# B&R Automation Studio project Panasonic_LinkaPowerCP2_A2021055 (part 4)

### Global.typ - Global data types
```iecst
(********************************************************************
 * COPYRIGHT -- Microsoft
 ********************************************************************
 * File: Global.typ
 * Author: Martin
 * Created: February 11, 2016
 ********************************************************************
 * Global data types of project Zamazat_1
 ********************************************************************)
(*************Vizualizacia******************************)

TYPE
	P1_Vizu_typ : 	STRUCT
		ActualPage : STRING[80];
		GoPage : STRING[80] := 'PageBootP1';
		TL_ResetCS : BOOL;
		TL_RezimAutomat : BOOL;
		ZobrazHL1_ST1 : BOOL; (*ST1 - Chýbajúci material na paletke 4F*)
		ZobrazHL2_ST1 : BOOL; (*ST1 - Chýbajúci material na paletke 5F*)
		ZobrazHL3_ST1 : BOOL; (*ST1 - Chýbajúci material na paletke 5H*)
		ZobrazHL4_ST1 : BOOL; (*ST1 - Zlý alebo neprečítaný QR kód na Power CP*)
		ZobrazHL5_ST1 : BOOL; (*ST1 - Zle zacvaknuté alebo chýbajúce piny DPS*)
		ZobrazHL6_ST1 : BOOL; (*ST1 - Zlý alebo neprečítaný QR kód DPS*)
		ZobrazHL7_ST1 : BOOL; (*ST1 - Nesprávny QR kód Power CP*)
		ZobrazHL8_ST1 : BOOL; (*ST1 - Nesprávny QR kód DPS*)
		ZobrazHL9_ST1 : BOOL; (*ST1 - Odpoved systemu tracebility je NG*)
		ZobrazHL10_ST1 : BOOL;
		ZobrazHL11_ST1 : BOOL;
		ZobrazHL12_ST1 : BOOL;
		ZobrazHL13_ST1 : BOOL;
		ZobrazHL14_ST1 : BOOL; (*ST1 - Nieje prihlásený operátor*)
		ZobrazHL15_ST1 : BOOL; (*ST1 - Panatrace neodpovedá*)
		ZobrazHL1_ST2 : BOOL;
		ZobrazHL2_ST2 : BOOL;
		ZobrazHL3_ST2 : BOOL;
		ZobrazHL4_ST2 : BOOL;
		ZobrazHL5_ST2 : BOOL;
		ZobrazHL6_ST2 : BOOL;
		ZobrazHL7_ST2 : BOOL;
		ZobrazHL8_ST2 : BOOL;
		ZobrazHL9_ST2 : BOOL; (*ST2 - Odpoved panatrace NG*)
		ZobrazHL10_ST2 : BOOL; (*ST2 - Panatrace neodpovedá*)
		TL_PrednyZamok_Farba : WSTRING[80];
		TL_ZadnyZamok_Farba : WSTRING[80];
		TL_ZamkniPrednyZamok : BOOL;
		TL_ZamkniZadnyZamok : BOOL;
		TL_StartAutomat_ENABLE : BOOL;
		TL_KoniecCyklu_ENABLE : BOOL;
		TL_Uzivatelia_ENABLE : BOOL;
		TL_STOP_ENABLE : BOOL;
		TL_SETUP_ENABLE : BOOL;
		TL_VyprazdnenieLinky_ENABLE : BOOL;
		TL_RezimAutomat_ENABLE : BOOL;
		TL_RezimManual_ENABLE : BOOL;
		TL_OvladaniaZamkov_ENABLE : BOOL;
		TL_VolbaModelu_ENABLE : BOOL;
		TL_PaletkaPrechadza_ENABLE : BOOL;
		TL_TestovaciKus_ENABLE : BOOL;
		TL_Revork_ENABLE : BOOL;
		TL_OvladanieVytahu_ENABLE : BOOL;
		TL_PrihlasenieOperatora_ENABLE : BOOL;
		TL_PrihlasovOperatora_AKTIVNE : BOOL;
		TL_VycistiSkrutkovackuK30_ENABLE : BOOL;
		TL_PolohujManipulator_ENABLE : BOOL;
		Tl_VysunutieSkrutkovK30_ENABLE : BOOL;
		TL_OvladaniaVysunSkrutkovM4_M5 : BOOL;
		TL_OvladSkrutkovSetuK30_ENABLE : BOOL;
		TL_OvladManipulatoraXY_ENABLE : BOOL;
		Srobovanie_OvlManipOsX_ENABLE : BOOL;
		Srobovanie_OvlManipOsY_ENABLE : BOOL;
		EditaciaParametrov_ENABLE : BOOL;
		RR_CistenieSkrutkovaciek_ENABLE : BOOL;
		RR_PozicieSkrutiek_ENABLE : BOOL;
		Vytah_CitaniePaletky_ENABLE : BOOL;
		Vytah_ZapisPaletky_ENABLE : BOOL;
		Warnings_Farba : WSTRING[80];
		Warnings_Index : USINT;
		IndexStavu_Dopravnik : USINT;
		IndexStavu_Vytah : USINT;
		IndexStavu_SpodnyStoper : USINT;
		IndexStavu_StoperSrobovania : USINT;
		IndexStavu_Srobovanie : USINT;
		IndexStavu_AkumulacnyStoper : USINT;
		IndexStavu_Robot : USINT;
	END_STRUCT;
	P2_Vizu_typ : 	STRUCT
		ActualPage : STRING[80];
		GoPage : STRING[80] := 'PageBootP2';
		TL_RezimAutomat : BOOL;
		TL_PrednyZamok_Farba : WSTRING[80];
		TL_ZadnyZamok_Farba : WSTRING[80];
		TL_ZamkniPredneZamky : BOOL;
		TL_ZamkniZadneZamky : BOOL;
		TL_StartAutomat_ENABLE : BOOL;
		TL_KoniecCyklu_ENABLE : BOOL;
		TL_STOP_ENABLE : BOOL;
		TL_SETUP_ENABLE : BOOL;
		TL_RezimAutomat_ENABLE : BOOL;
		TL_RezimManual_ENABLE : BOOL;
		TL_RRZdvihZaklTesnenia_ENABLE : BOOL;
		TL_RRPojazdZaklTesnenia_ENABLE : BOOL;
		TL_OvladaniaZamkov_ENABLE : BOOL;
		TL_VycistiSkrutkovackuM6_ENABLE : BOOL;
		TL_VycistiSkrutkovackuM5_ENABLE : BOOL;
		TL_PolohujManipulator_ENABLE : BOOL;
		TL_VysunutiaMaticovacM4_ENABLE : BOOL;
		Tl_VysunutieSkrutkovM6_ENABLE : BOOL;
		Tl_VysunutieSkrutkovM5_ENABLE : BOOL;
		TL_OvladaniaVysunSkrutkovM4 : BOOL;
		TL_OvladManipulatoraXY_ENABLE : BOOL;
		TL_OvladSkrutkovSetuM6_ENABLE : BOOL;
		TL_OvladSkrutkovSetuM5_ENABLE : BOOL;
		TL_PresunZvarania_ENABLE : BOOL;
		TL_ZdvihZvarania_ENABLE : BOOL;
		TL_StartSekvencieZvarania_ENABLE : BOOL;
		EditaciaParametrov_ENABLE : BOOL;
		ZaklTesnenia_OvlZdvihu_ENABLE : BOOL;
		ZaklTesnenia_OvlZostupu_ENABLE : BOOL;
		ZaklTesnenia_OvlPojazdu_ENABLE : BOOL;
		Srobovanie_OvlManipOsX_ENABLE : BOOL;
		Srobovanie_OvlManipOsY_ENABLE : BOOL;
		Zvaranie_OvlZdvihu_ENABLE : BOOL;
		RR_CistenieSkrutkovaciek_ENABLE : BOOL;
		RR_PozicieSkrutiek_ENABLE : BOOL;
		TL_PrihlasenieOperatora_ENABLE : BOOL;
		TL_PrihlasovOperatora_AKTIVNE : BOOL;
		TL_ResetCS : BOOL;
		Warnings_Farba : WSTRING[80];
		Warnings_Index : USINT;
		StavPracoviska_Index : USINT;
		ZobrazPopUp_0 : BOOL;
		ZobrazPopUp_1 : BOOL;
		ZobrazPopUp_2 : BOOL;
		PopUpButtonYES : BOOL;
		PopUpButtonNO : BOOL;
		ZobrazHL1_ST3 : BOOL; (*ST3 - Chýbajúci material na paletke 4F *)
		ZobrazHL2_ST3 : BOOL; (*ST3 - Chýbajúci material na paletke 5F*)
		ZobrazHL3_ST3 : BOOL; (*ST3 - Chýbajúci material na paletke 5H*)
		ZobrazHL4_ST3 : BOOL; (*ST3 - Skontroluj prítomnosť alebo QR kód filtra 5H*)
		ZobrazHL5_ST3 : BOOL; (*ST3 - V zakladači chýba Power CP !!!*)
		ZobrazHL6_ST3 : BOOL; (*ST3 - V zakladači chýba tesnenie !!!*)
		ZobrazHL7_ST3 : BOOL; (*ST3 - Zle založené tesnenie na Power CP*)
		ZobrazHL8_ST3 : BOOL; (*ST3 - Založenie tesnenia je OK, odober Power CP zo zakladača *)
		ZobrazHL9_ST3 : BOOL; (*ST3 - Nesprávny QR kód filtra 5H*)
		ZobrazHL10_ST3 : BOOL; (*ST3 - Nesprávny alebo neprečítaný QR kód Power CP*)
		ZobrazHL11_ST3 : BOOL; (*ST3 - Odpoved systemu tracebility je NG*)
		ZobrazHL12_ST3 : BOOL; (*ST3 - Operátor nieje prihlásený*)
		ZobrazHL13_ST3 : BOOL; (*ST3 - Odpoved panatrace je NG*)
		ZobrazHL14_ST3 : BOOL; (*ST3 - Odober PowerCP z paletky a vlož do šuplíka*)
		ZobrazHL15_ST3 : BOOL; (*ST3 - Panatrace neodpovedá*)
		ZobrazHL1_ST4 : BOOL;
		ZobrazHL2_ST4 : BOOL;
		ZobrazHL3_ST4 : BOOL; (*ST4 -Odpoved panatrace je NG*)
		ZobrazHL4_ST4 : BOOL; (*ST4 - Panatrace neodpovedá*)
		ZobrazHL1_ST5 : BOOL;
		ZobrazHL2_ST5 : BOOL;
		ZobrazHL3_ST5 : BOOL;
		ZobrazHL4_ST5 : BOOL; (*ST5 - Odpoved panatrace je NG*)
		ZobrazHL5_ST5 : BOOL; (*ST5 - Model 4F kontrola skrutiek M4 s komaxitom*)
		ZobrazHL6_ST5 : BOOL; (*ST5 - Model 5F kontrola skrutiek M4 s komaxitom*)
		ZobrazHL7_ST5 : BOOL; (*ST5 - Model 5H kontrola skrutiek M4 bez komaxitu*)
		ZobrazHL8_ST5 : BOOL; (*ST5 - Panatrace neodpovedá*)
		ZobrazHL1_ST6 : BOOL; (*ST6 - Chýbajúci material na paletke 4F *)
		ZobrazHL2_ST6 : BOOL; (*ST6 - Chýbajúci material na paletke 5F*)
		ZobrazHL3_ST6 : BOOL; (*ST6 - Chýbajúci material na paletke 5H*)
		ZobrazHL4_ST6 : BOOL; (*ST6 - Skontroluj prítomnosť alebo QR kód filtra 5H*)
		ZobrazHL5_ST6 : BOOL; (*ST6 - V zakladači chýba Power CP !!!*)
		ZobrazHL6_ST6 : BOOL; (*ST6 - V zakladači chýba tesnenie !!!*)
		ZobrazHL7_ST6 : BOOL; (*ST6 - Zle založené tesnenie na Power CP*)
		ZobrazHL8_ST6 : BOOL; (*ST6 - Odpoved panatrace je NG*)
		ZobrazHL9_ST6 : BOOL; (*ST6 - Panatrace neodpovedá*)
		IndexStavu_Dopravnik : USINT;
		IndexStavu_SpodnyStoper : USINT;
		IndexStavu_StoperZakladacaTesn : USINT;
		IndexStavu_ZakladacaTesnenia : USINT;
		IndexStavu_StoperMaticovacky : USINT;
		IndexStavu_AkumulacnyStoper : USINT;
		IndexStavu_StoperSrobovania : USINT;
		IndexStavu_Srobovania : USINT;
		IndexStavu_Robot : USINT;
		IndexStavu_StoperZvarania : USINT;
		IndexStavu_Zvaranie : USINT;
		IndexStavu_Cistenie : USINT;
	END_STRUCT;
	P34_Vizu_typ : 	STRUCT
		ActualPage : STRING[80];
		GoPage : STRING[80] := 'PageBootP34';
		TL_RezimAutomat : BOOL;
		ZobrazHL1_ST7 : BOOL; (*ST7 - Odpoved panatrace je NG*)
		ZobrazHL2_ST7 : BOOL; (*ST7 - Panatrace neodpovedá*)
		ZobrazHL1_ST8 : BOOL; (*ST8A - Odpoved panatrace je NG*)
		ZobrazHL2_ST8 : BOOL; (*ST8B - Odpoved panatrace je NG*)
		ZobrazHL3_ST8 : BOOL; (*ST8A - Panatrace neodpovedá*)
		ZobrazHL4_ST8 : BOOL; (*ST8B - Panatrace neodpovedá*)
		ZobrazHL1_ST9 : BOOL;
		ZobrazHL2_ST9 : BOOL;
		ZobrazHL3_ST9 : BOOL; (*ST9 - Odpoved panatrace je NG*)
		ZobrazHL4_ST9 : BOOL; (*ST9 - Panatrace neodpovedá*)
		ZobrazHL1_ST10 : BOOL; (*ST10 - Chýbajúci material na paletke 4F *)
		ZobrazHL2_ST10 : BOOL; (*ST10 - Chýbajúci material na paletke 5F*)
		ZobrazHL3_ST10 : BOOL; (*ST10 - Chýbajúci material na paletke 5H*)
		ZobrazHL4_ST10 : BOOL; (*ST10 - Paletka nieje prázdna*)
		ZobrazHL5_ST10 : BOOL; (*ST10 - Paletka nieje prázdna*)
		ZobrazHL6_ST10 : BOOL; (*ST10 - Paletka nieje prázdna*)
		ZobrazHL7_ST10 : BOOL; (*ST10 - Nieje prihlaseny operator*)
		ZobrazHL8_ST10 : BOOL;
		ZobrazHL9_ST10 : BOOL; (*ST10 - Odpoved panatrace je NG*)
		ZobrazHL10_ST10 : BOOL; (*ST10 - Panatrace neodpovedá*)
		ZobrazHL1_HVtest : BOOL; (*HV tester neodpovedá*)
		ZobrazHL1_FinalTestA : BOOL; (*Final tester neodpovedá*)
		ZobrazHL1_FinalTestB : BOOL; (*Final tester neodpovedá*)
		TL_ResetCS : BOOL;
		IndexStavu_DopravnikP3 : USINT;
		IndexStavu_SpodnyStoperP3 : USINT;
		IndexStavu_StoperSrobovaniaP3 : USINT;
		IndexStavu_SrobovanieP3 : USINT;
		IndexStavu_HV_Test : USINT;
		IndexStavu_AkumulacnyStoperP3 : USINT;
		IndexStavu_ZdvizkPredLeakTestomA : USINT;
		IndexStavu_ZdvizkPredLeakTestomB : USINT;
		IndexStavu_StoperLeakageTestA : USINT;
		IndexStavu_StoperLeakageTestB : USINT;
		IndexStavu_ZdvizkaZaLeakTestomA : USINT;
		IndexStavu_ZdvizkaZaLeakTestomB : USINT;
		IndexStavu_DopravnikP4 : USINT;
		IndexStavu_SpodnyStoperP4 : USINT;
		IndexStavu_Vytah : USINT;
		IndexStavu_StoperFunkcnyTestA : USINT;
		IndexStavu_StoperFunkcnyTestB : USINT;
		IndexStavu_ZdvizkaZaFunkTestomA : USINT;
		IndexStavu_ZdvizkaZaFunkTestomB : USINT;
		IndexStavu_StoperEtiketovackyP4 : USINT;
		TL_PrednyZamok_Farba_P3 : WSTRING[80];
		TL_ZadnyZamok_Farba_P3 : WSTRING[80];
		TL_ZamkniPredneZamky_P3 : BOOL;
		TL_ZamkniZadneZamky_P3 : BOOL;
		TL_StartAutomat_ENABLE_P3 : BOOL;
		TL_KoniecCyklu_ENABLE_P3 : BOOL;
		TL_STOP_ENABLE_P3 : BOOL;
		TL_SETUP_ENABLE : BOOL;
		TL_RezimAutomat_ENABLE : BOOL;
		TL_RezimManual_ENABLE_P3 : BOOL;
		TL_RezimManual_ENABLE_P4 : BOOL;
		TL_OvladaniaZamkov_ENABLE_P3 : BOOL;
		TL_OvladaniaZamkov_ENABLE_P4 : BOOL;
		TL_StartAutomat_ENABLE_P4 : BOOL;
		TL_KoniecCyklu_ENABLE_P4 : BOOL;
		TL_STOP_ENABLE_P4 : BOOL;
		TL_VycistiSkrutkovackuK40_ENABLE : BOOL;
		TL_PolohujManipulator_ENABLE : BOOL;
		Tl_VysunutieSkrutkovK40_ENABLE : BOOL;
		TL_OvladaniaVysunSkrutkovM5 : BOOL;
		TL_OvladManipulatoraY_ENABLE : BOOL;
		TL_OvladSkrutkovSetuK40_ENABLE : BOOL;
		TL_SekvencieHV_Testu_ENABLE : BOOL;
		TL_OvladaniaHV_Testu_ENABLE : BOOL;
		TL_SekvencieLeakTestuA_ENABLE : BOOL;
		TL_OvladaniaLeakTestuA_ENABLE : BOOL;
		TL_SekvencieLeakTestuB_ENABLE : BOOL;
		TL_OvladaniaLeakTestuB_ENABLE : BOOL;
		TL_SekvencieFunkcTestuA_ENABLE : BOOL;
		TL_OvladaniaFunkcTestuA_ENABLE : BOOL;
		TL_SekvencieFunkcTestuB_ENABLE : BOOL;
		TL_OvladaniaFunkcTestuB_ENABLE : BOOL;
		TL_SekvencieEtiketovania_ENABLE : BOOL;
		TL_OvladaniaEtiketovania_ENABLE : BOOL;
		TL_ZdvihAplikEtiketovania_ENABLE : BOOL;
		Vytah_CitaniePaletky_ENABLE : BOOL;
		Vytah_ZapisPaletky_ENABLE : BOOL;
		Srobovanie_OvlManipOsY_ENABLE : BOOL;
		VolbaLeakageTestu_ENABLE : BOOL;
		VolbaFunkcnehoTestu_ENABLE : BOOL;
		EditaciaParametrov_ENABLE : BOOL;
		RR_CistenieSkrutkovaciek_ENABLE : BOOL;
		RR_PozicieSkrutiek_ENABLE : BOOL;
		TL_PrihlasenieOperatora_ENABLE : BOOL;
		TL_PrihlasovOperatora_AKTIVNE : BOOL;
		TL_PrednyZamok_Farba_P4 : WSTRING[80];
		TL_ZadnyZamok_Farba_P4 : WSTRING[80];
		TL_ZamkniPrednyZamok_P4 : BOOL;
		TL_ZamkniZadnyZamok_P4 : BOOL;
		WarningsP3_Farba : WSTRING[80];
		WarningsP3_Index : USINT;
		WarningsP4_Farba : WSTRING[80];
		WarningsP4_Index : USINT;
		TL_VyprazdnenieLinky_ENABLE : BOOL;
	END_STRUCT;
	Vizu_typ : 	STRUCT
		TL_ResetCS_Farba : WSTRING[80];
		ZadanyCasPLC : DATE_AND_TIME;
		NastavCasPLC : BOOL;
		AktualnyCasPLC : DATE_AND_TIME;
	END_STRUCT;
END_TYPE

(*************Parametre paletky*********************)

TYPE
	Paletka_typ : 	STRUCT
		PAR : Paletka_PAR_typ; (*Parametre komunikácie z Panatrace*)
		STAV : Paletka_STAV_typ;
	END_STRUCT;
	Paletka_PAR_typ : 	STRUCT
		CisloPaletky : STRING[2]; (*Je pevne dané čipom RFID*)
		QRkodPowerCP : STRING[30]; (*Načítam ho na prvom výťahu a posielam ho na server ako master number *)
		QRkodFiltra_5H : STRING[32]; (*Načítam ho na pracovisku zakladania tesnenia a párujem ho s QR kodom Power CP*)
		QRkodFiltra_4F5F : STRING[32]; (*Načítam ho na prvom výtahu a párujem ho s QR kodom Power CP*)
		ID_Operatora : STRING[80]; (*Číslo karty operátora*)
		StavPowerCP : STRING[4]; (*Stav vyžiadaný zo servera  - PASS, FAIL,  ktorý sa mení v pribehu výroby *)
	END_STRUCT;
	Paletka_STAV_typ : 	STRUCT
		StavPaletky : STRING[10]; (*OK - paletka OK , NG - paletka NG, REV - revork, TEST - testovací kus, PRECH - paletka iba prechádza*)
		TypModelu : STRING[5]; (*4F, 5F, 5H podla zvolenej receptury*)
		KodModelu : STRING[32]; (*Dostanem pridelene na pracovisku etiketovania*)
		CisloTestovacejStanice : STRING[20]; (*Číslo testovacej stanice*)
		CisloRevorkovejStanice : STRING[20]; (*Číslo revorkovej stanice*)
		Zvaranie_Ukoncene : BOOL;
		HV_Test_Ukonceny : BOOL;
		LeakageTest_Ukonceny : BOOL;
		FunkcnyTest_Ukonceny : BOOL;
		QRkodFiltraPriradeny : BOOL;
		NalepenieEtikety_DONE : BOOL;
		OdoslanieFotiek_DONE : BOOL;
		Komunikacia_DONE : BOOL;
		CisloEtiketyVyziadane : BOOL;
	END_STRUCT;
END_TYPE

(*****************Remanentne premenne**********)

TYPE
	P1_RemPremenne_typ : 	STRUCT
		P1_Srob45F_PozX_LavejSkrutkyK30 : REAL;
		P1_Srob45F_PozY_LavejSkrutkyK30 : REAL;
		P1_Srob45F_PozX_PravejSkrutkyK30 : REAL;
		P1_Srob45F_PozY_PravejSkrutkyK30 : REAL;
		P1_Srob4F_PozX_ZadnejSkrutkyM4 : REAL;
		P1_Srob4F_PozY_ZadnejSkrutkyM4 : REAL;
		P1_Srob5F_PozX_ZadnejSkrutkyM4 : REAL;
		P1_Srob5F_PozY_ZadnejSkrutkyM4 : REAL;
		P1_Srob45F_Mom_ZadnejSkrutkyM4 : REAL;
		P1_Srob45F_Rychl_ZadnejSkrutkyM4 : REAL; (*mm/s*)
		P1_Srob4F_PozX_PrednejSkrutkyM4 : REAL;
		P1_Srob4F_PozY_PrednejSkrutkyM4 : REAL;
		P1_Srob5F_PozX_PrednejSkrutkyM4 : REAL;
		P1_Srob5F_PozY_PrednejSkrutkyM4 : REAL;
		P1_Srob45F_Mom_PrednejSkrutkyM4 : REAL;
		P1_Srob45F_Rychl_PredneSkrutkyM4 : REAL; (*mm/s*)
		P1_Srob45F_PozX_SkrutkyDPS_M4 : REAL;
		P1_Srob45F_PozY_SkrutkyDPS_M4 : REAL;
		P1_Srob45F_Mom_SkrutkyDPS_M4 : REAL;
		P1_Srob45F_Rychl_SkrutkyDPS_M4 : REAL; (*mm/s*)
		P1_Srob5H_PozX_LavejSkrutkyK30 : REAL;
		P1_Srob5H_PozY_LavejSkrutkyK30 : REAL;
		P1_Srob5H_PozX_PravejSkrutkyK30 : REAL;
		P1_Srob5H_PozY_PravejSkrutkyK30 : REAL;
		P1_Srob5H_PozX_LavejSkrutkyM5 : REAL;
		P1_Srob5H_PozY_LavejSkrutkyM5 : REAL;
		P1_Srob5H_Mom_LavejSkrutkyM5 : REAL;
		P1_Srob5H_Rychl_LavejSkrutkyM5 : REAL; (*mm/s*)
		P1_Srob5H_PozX_StrednejSkrutkyM5 : REAL;
		P1_Srob5H_PozY_StrednejSkrutkyM5 : REAL;
		P1_Srob5H_Mom_StrednejSkrutkyM5 : REAL;
		P1_Srob5H_Rychl_StredneSkrutkyM5 : REAL; (*mm/s*)
		P1_Srob5H_PozX_PravejSkrutkyM5 : REAL;
		P1_Srob5H_PozY_PravejSkrutkyM5 : REAL;
		P1_Srob5H_Mom_PravejSkrutkyM5 : REAL;
		P1_Srob5H_Rychl_PravejSkrutkyM5 : REAL; (*mm/s*)
		P1_Srob_PozX_OdobratSkrutkyM5 : REAL;
		P1_Srob_PozY_OdobratSkrutkyM5 : REAL;
		P1_Srob_PozZ_OdobratSkrutkyM5 : REAL;
		P1_Srob_PozX_OdobratSkrutkyM4 : REAL;
		P1_Srob_PozY_OdobratSkrutkyM4 : REAL;
		P1_Srob_PozZ_OdobratSkrutkyM4 : REAL;
		P1_Vytah_RychlostZdvihu : REAL; (*mm/s*)
		P1_Vytah_Zdvih_Acc : REAL;
		P1_Vytah_Zdvih_Dcc : REAL;
		P1_Vytah_PoziciaNakladania : REAL;
		P1_Vytah_PoziciaVykladania : REAL;
		P1_ManipSrob_OsX_Rychlost : REAL; (*mm/s*)
		P1_ManipSrob_OsY_Rychlost : REAL; (*mm/s*)
		P1_ManipSrob_OsXY_Acc : REAL;
		P1_ManipSrob_OsXY_Dcc : REAL;
		P1_ManipSrob_OsZ_M4_Rychlost : REAL; (*mm/s*)
		P1_ManipSrob_OsZ_M4_Acc : REAL;
		P1_ManipSrob_OsZ_M4_Dcc : REAL;
		P1_ManipSrob_OsZ_M5_Rychlost : REAL; (*mm/s*)
		P1_ManipSrob_OsZ_M5_Acc : REAL;
		P1_ManipSrob_OsZ_M5_Dcc : REAL;
		P1_Srob45F_LavaK30_Vysunutie_LO : REAL; (*Vysunutie skrutkovačky - spodná tolerancia*)
		P1_Srob45F_LavaK30_Vysunutie_HI : REAL; (*Vysunutie skrutkovačky - horná tolerancia*)
		P1_Srob45F_PravaK30_Vysunutie_LO : REAL; (*Vysunutie skrutkovačky - spodná tolerancia*)
		P1_Srob45F_PravaK30_Vysunutie_HI : REAL; (*Vysunutie skrutkovačky - horná tolerancia*)
		P1_Srob45F_ZadnaM4_Vysunutie_LO : REAL; (*Vysunutie skrutkovačky - spodná tolerancia*)
		P1_Srob45F_ZadnaM4_Vysunutie_HI : REAL; (*Vysunutie skrutkovačky - horná tolerancia*)
		P1_Srob45F_PrednaM4_Vysunutie_LO : REAL; (*Vysunutie skrutkovačky - spodná tolerancia*)
		P1_Srob45F_PrednaM4_Vysunutie_HI : REAL; (*Vysunutie skrutkovačky - horná tolerancia*)
		P1_Srob45F_DPS_M4_Vysunutie_LO : REAL; (*Vysunutie skrutkovačky - spodná tolerancia*)
		P1_Srob45F_DPS_M4_Vysunutie_HI : REAL; (*Vysunutie skrutkovačky - horná tolerancia*)
		P1_Srob5H_LavaK30_Vysunutie_LO : REAL; (*Vysunutie skrutkovačky - spodná tolerancia*)
		P1_Srob5H_LavaK30_Vysunutie_HI : REAL; (*Vysunutie skrutkovačky - horná tolerancia*)
		P1_Srob5H_PravaK30_Vysunutie_LO : REAL; (*Vysunutie skrutkovačky - spodná tolerancia*)
		P1_Srob5H_PravaK30_Vysunutie_HI : REAL; (*Vysunutie skrutkovačky - horná tolerancia*)
		P1_Srob5H_LavaM5_Vysunutie_LO : REAL; (*Vysunutie skrutkovačky - spodná tolerancia*)
		P1_Srob5H_LavaM5_Vysunutie_HI : REAL; (*Vysunutie skrutkovačky - horná tolerancia*)
		P1_Srob5H_StrednaM5_Vysunutie_LO : REAL; (*Vysunutie skrutkovačky - spodná tolerancia*)
		P1_Srob5H_StrednaM5_Vysunutie_HI : REAL; (*Vysunutie skrutkovačky - horná tolerancia*)
		P1_Srob5H_PravaM5_Vysunutie_LO : REAL; (*Vysunutie skrutkovačky - spodná tolerancia*)
		P1_Srob5H_PravaM5_Vysunutie_HI : REAL; (*Vysunutie skrutkovačky - horná tolerancia*)
	END_STRUCT;
	P2_RemPremenne_typ : 	STRUCT
		P2_ZaklTesn_Zdvih_RychlostZdvihu : REAL; (*mm/s*)
		P2_ZaklTesn_Zdvih_RychlZatlacen : REAL; (*mm/s*)
		P2_ZaklTesn_Zdvih_Acc : REAL;
		P2_ZaklTesn_Zdvih_Dcc : REAL;
		P2_ZaklTesn_Zdvih_MomZatlacen : REAL;
		P2_ZaklTesn_Zdvih_PozZatlacenia : REAL;
		P2_ZaklTesn_Pojazd_RychlVysun : REAL;
		P2_ZaklTesn_Pojazd_RychlZasun : REAL;
		P2_ZaklTesn_Pojazd_Acc : REAL;
		P2_ZaklTesn_Pojazd_Dcc : REAL;
		P2_ZaklTesn_Pojazd_PozZatlacenia : REAL;
		P2_ZaklTesn_Pojazd_PozVkladania : REAL;
		P2_ZaklTesn_PocetZatlaceni : USINT;
		P2_Srob4F_PozX_LavejSkrutkyM6 : REAL;
		P2_Srob4F_PozY_LavejSkrutkyM6 : REAL;
		P2_Srob4F_PozX_PravejSkrutkyM6 : REAL;
		P2_Srob4F_PozY_PravejSkrutkyM6 : REAL;
		P2_Srob4F_PozX_LavejSkrutkyM4 : REAL;
		P2_Srob4F_PozY_LavejSkrutkyM4 : REAL;
		P2_Srob45F_Mom_LavejSkrutkyM4 : REAL;
		P2_Srob45F_Rychl_LavejSkrutkyM4 : REAL; (*mm/s*)
		P2_Srob4F_PozX_PravejSkrutkyM4 : REAL;
		P2_Srob4F_PozY_PravejSkrutkyM4 : REAL;
		P2_Srob45F_Mom_PravejSkrutkyM4 : REAL;
		P2_Srob45F_Rychl_PravejSkrutkyM4 : REAL; (*mm/s*)
		P2_Srob5F_PozX_LavejSkrutkyM6 : REAL;
		P2_Srob5F_PozY_LavejSkrutkyM6 : REAL;
		P2_Srob5F_PozX_PravejSkrutkyM6 : REAL;
		P2_Srob5F_PozY_PravejSkrutkyM6 : REAL;
		P2_Srob5F_PozX_LavejSkrutkyM4 : REAL;
		P2_Srob5F_PozY_LavejSkrutkyM4 : REAL;
		P2_Srob5F_PozX_PravejSkrutkyM4 : REAL;
		P2_Srob5F_PozY_PravejSkrutkyM4 : REAL;
		P2_Srob5H_PozX_LavejSkrutkyM5 : REAL;
		P2_Srob5H_PozY_LavejSkrutkyM5 : REAL;
		P2_Srob5H_PozX_PravejSkrutkyM5 : REAL;
		P2_Srob5H_PozY_PravejSkrutkyM5 : REAL;
		P2_Srob5H_PozX_SkrutkyM4 : REAL;
		P2_Srob5H_PozY_SkrutkyM4 : REAL;
		P2_Srob5H_Mom_SkrutkyM4 : REAL;
		P2_Srob5H_Rychl_SkrutkyM4 : REAL; (*mm/s*)
		P2_Srob_PozX_OdobratSkrutkyM4 : REAL;
		P2_Srob_PozY_OdobratSkrutkyM4 : REAL;
		P2_Srob_PozZ_OdobratSkrutkyM4 : REAL;
		P2_ManipSrob_OsX_Rychlost : REAL;
		P2_ManipSrob_OsY_Rychlost : REAL;
		P2_ManipSrob_OsX_Acc : REAL;
		P2_ManipSrob_OsX_Dcc : REAL;
		P2_ManipSrob_OsY_Acc : REAL;
		P2_ManipSrob_OsY_Dcc : REAL;
		P2_ManipSrob_OsZ_M4_Rychlost : REAL; (*mm/s*)
		P2_ManipSrob_OsZ_M4_Acc : REAL;
		P2_ManipSrob_OsZ_M4_Dcc : REAL;
		P2_Zvaranie_MomentZvarania_PS : REAL;
		P2_Zvaranie_MomentZvarania_LS : REAL;
		P2_Zvaranie_RychlostZvarania : REAL; (*mm/s*)
		P2_Zvaranie_Acc : REAL;
		P2_Zvaranie_Dcc : REAL;
		P2_Zvaranie_PoziciaZvarania_PS : REAL;
		P2_Zvaranie_PoziciaZvarania_LS : REAL;
		P2_Zvaranie_CasZvarania : TIME;
		P2_Zvaranie_RychlostZdvihu : REAL; (*mm/s*)
		P2_Srob45F_LavaM6_Vysunutie_LO : REAL; (*Vysunutie skrutkovačky - spodná tolerancia*)
		P2_Srob45F_LavaM6_Vysunutie_HI : REAL; (*Vysunutie skrutkovačky - horná tolerancia*)
		P2_Srob45F_PravaM6_Vysunutie_LO : REAL; (*Vysunutie skrutkovačky - spodná tolerancia*)
		P2_Srob45F_PravaM6_Vysunutie_HI : REAL; (*Vysunutie skrutkovačky - horná tolerancia*)
		P2_Srob45F_LavaM4_Vysunutie_LO : REAL; (*Vysunutie skrutkovačky - spodná tolerancia*)
		P2_Srob45F_LavaM4_Vysunutie_HI : REAL; (*Vysunutie skrutkovačky - horná tolerancia*)
		P2_Srob45F_PravaM4_Vysunutie_LO : REAL; (*Vysunutie skrutkovačky - spodná tolerancia*)
		P2_Srob45F_PravaM4_Vysunutie_HI : REAL; (*Vysunutie skrutkovačky - horná tolerancia*)
		P2_Srob5H_LavaM5_Vysunutie_LO : REAL; (*Vysunutie skrutkovačky - spodná tolerancia*)
		P2_Srob5H_LavaM5_Vysunutie_HI : REAL; (*Vysunutie skrutkovačky - horná tolerancia*)
		P2_Srob5H_PravaM5_Vysunutie_LO : REAL; (*Vysunutie skrutkovačky - spodná tolerancia*)
		P2_Srob5H_PravaM5_Vysunutie_HI : REAL; (*Vysunutie skrutkovačky - horná tolerancia*)
		P2_Srob5H_StrednaM4_Vysunutie_LO : REAL; (*Vysunutie skrutkovačky - spodná tolerancia*)
		P2_Srob5H_StrednaM4_Vysunutie_HI : REAL; (*Vysunutie skrutkovačky - horná tolerancia*)
		P2_Maticovacka_Vysunutie_LO : REAL; (*Vysunutie skrutkovačky - spodná tolerancia*)
		P2_Maticovacka_Vysunutie_HI : REAL; (*Vysunutie skrutkovačky - horná tolerancia*)
		P2_Zvaranie_MomentZatlacania : REAL;
		P2_Zvaranie_RychlostZatlacania : REAL; (*mm/s*)
		P2_Zvaranie_CasZatlacania : TIME;
	END_STRUCT;
	P34_RemPremenne_typ : 	STRUCT
		P3_ManipSrob_OsY_Rychlost : REAL; (*mm/s*)
		P3_ManipSrob_OsY_Acc : REAL;
		P3_ManipSrob_OsY_Dcc : REAL;
		P3_ManipSrob_OsZ_M5_Rychlost : REAL; (*mm/s*)
		P3_ManipSrob_OsZ_M5_Acc : REAL;
		P3_ManipSrob_OsZ_M5_Dcc : REAL;
		P3_Srob45F_PozY_Skrutkovania : REAL;
		P3_Srob5H_PozY_Skrutkovania : REAL;
		P3_Srob_PozY_OdobratSkrutkyM5 : REAL;
		P3_Srob_PozZ_OdobratSkrutkyM5 : REAL;
		P3_Srob45F_Mom_SkrutkyM5 : REAL;
		P3_Srob45F_Rychl_SkrutkyM5 : REAL; (*mm/s*)
		P3_Srob5H_Mom_SkrutkyM5 : REAL;
		P3_Srob5H_Rychl_SkrutkyM5 : REAL; (*mm/s*)
		P3_Srob45F_K40_Vysunutie_LO : REAL; (*Vysunutie skrutkovačky - spodná tolerancia*)
		P3_Srob45F_K40_Vysunutie_HI : REAL; (*Vysunutie skrutkovačky - horná tolerancia*)
		P3_Srob45F_M5_Vysunutie_LO : REAL; (*Vysunutie skrutkovačky - spodná tolerancia*)
		P3_Srob45F_M5_Vysunutie_HI : REAL; (*Vysunutie skrutkovačky - horná tolerancia*)
		P3_Srob5H_M5_Vysunutie_LO : REAL; (*Vysunutie skrutkovačky - spodná tolerancia*)
		P3_Srob5H_M5_Vysunutie_HI : REAL; (*Vysunutie skrutkovačky - horná tolerancia*)
		P4_Vytah_RychlostZdvihu : REAL; (*mm/s*)
		P4_Vytah_Zdvih_Acc : REAL;
		P4_Vytah_Zdvih_Dcc : REAL;
		P4_Vytah_PoziciaNakladania : REAL;
		P4_Vytah_PoziciaVykladania : REAL;
		P4_ZdvihEtiketovacky_Acc : REAL;
		P4_ZdvihEtiketovacky_Dcc : REAL;
		P4_Etiketov_RychlZdvihuAplikat : REAL; (*mm/s*)
		P4_Etiketovacka_PozOdoberEtikety : REAL;
		P4_Etiketovacka_PozEtikety_4F : REAL;
		P4_Etiketovacka_PozEtikety_5F : REAL;
		P4_Etiketovacka_PozEtikety_5H : REAL;
	END_STRUCT;
END_TYPE

(************************************Safety***********************************************************)

TYPE
	Safety_typ : 	STRUCT
		IN : Safety_IN_typ;
		OUT : Safety_OUT_typ;
		STAV : Safety_STAV_typ;
		Mapping_BYTE_IN : ARRAY[0..29]OF USINT;
		Mapping_BYTE_OUT : ARRAY[0..3]OF USINT;
	END_STRUCT;
	Safety_IN_typ : 	STRUCT
		Linka_SV_ZonaCS : BOOL;
		P1_SV_PrivodVzduchu_CH1 : BOOL;
		P1_SV_PrivodVzduchu_CH2 : BOOL;
		P1_SV_ZonaBunky : BOOL;
		P1_SV_ZonaVytahu : BOOL;
		P2_SV_PrivodVzduchu_CH1 : BOOL;
		P2_SV_PrivodVzduchu_CH2 : BOOL;
		P2_SV_ZonaBunky : BOOL;
		P2_SV_ZonaZakladacaTesnenia : BOOL;
		P2_SV_ZonaMaticovacky : BOOL;
		P2_SV_ZonaAutostopRobota : BOOL;
		P3_SV_PrivodVzduchu_CH1 : BOOL;
		P3_SV_PrivodVzduchu_CH2 : BOOL;
		P3_SV_ZonaBunky : BOOL;
		P3_SV_HV_test : BOOL;
		P4_SV_PrivodVzduchu_CH1 : BOOL;
		P4_SV_PrivodVzduchu_CH2 : BOOL;
		P4_SV_ZonaBunky : BOOL;
		P4_SV_ZonaVytahu : BOOL;
	END_STRUCT;
	Safety_OUT_typ : 	STRUCT
		Linka_ResetCS : BOOL;
		P1_ResetZonyVytahu : BOOL;
		P1_ResetZonyBunky : BOOL;
		P2_ResetZonyBunky : BOOL;
		P3_ResetZonyBunky : BOOL;
		P3_ResetZonyHVtest : BOOL;
		P4_ResetZonyBunky : BOOL;
		P4_ResetZonyVytahu : BOOL;
	END_STRUCT;
	Safety_STAV_typ : 	STRUCT
		Linka_SafetyPLC_Nabehlo : BOOL;
		Linka_ZonaCS_AKTIVNA : BOOL;
		Linka_TlacitkaCS_ODBLOKOVANE : BOOL;
		P1_Panel_TlacitkoCS_ODBLOK : BOOL;
		P1_Robot_TlacitkoCS_ODBLOK : BOOL;
		P1_Rozvadzac_TlacitkoCS_ODBLOK : BOOL;
		P1_VyblokovanieZamkov_AKTIVNE : BOOL;
		P1_Vytah_Bariera_AKTIVNA : BOOL;
		P1_Vytah_Muting_AKTIVNY : BOOL;
		P1_Bunka_Zamky_AKTIVNE : BOOL;
		P1_VstupBunky_VstupBar_AKTIVNA : BOOL;
		P1_VstupBunky_VystupBar_AKTIVNA : BOOL;
		P1_VystupBunky_VstupBar_AKTIVNA : BOOL;
		P1_VystupBunky_VystupBar_AKTIVNA : BOOL;
		P1_ZonaVytahu_AKTIVNA : BOOL;
		P1_ZonaBunky_AKTIVNA : BOOL;
		P1_DeadMan_AKTIVNY : BOOL;
		P2_Panel_TlacitkoCS_ODBLOK : BOOL;
		P2_Robot_TlacitkoCS_ODBLOK : BOOL;
		P2_DvojrucOvl_TlacitkoCS_ODBLOK : BOOL;
		P2_VyblokovanieZamkov_AKTIVNE : BOOL;
		P2_Rozvadzac_TlacitkoCS_ODBLOK : BOOL;
		P2_DeadMan_AKTIVNY : BOOL;
		P2_ZaklTesn_PojazdMuting_AKTIVNY : BOOL;
		P2_ZaklTesn_Bariera_AKTIVNA : BOOL;
		P2_ZaklTesn_Bumper_AKTIVNY : BOOL;
		P2_Bunka_VstupBariera_AKTIVNA : BOOL;
		P2_Bunka_Zamky_AKTIVNE : BOOL;
		P2_ZonaZakladacaPojazd_AKTIVNA : BOOL;
		P2_ZonaZakladacaZdvih_AKTIVNA : BOOL;
		P2_ZonaMaticovacky_AKTIVNA : BOOL;
		P2_DvojrucneOvladanie_AKTIVNE : BOOL;
		P2_ZonaBunky_AKTIVNA : BOOL;
		P3_VyblokovanieZamkov_AKTIVNE : BOOL;
		P3_Rozvadzac_TlacitkoCS_ODBLOK : BOOL;
		P3_DeadMan_AKTIVNY : BOOL;
		P3_Bunka_VstupBariera_AKTIVNA : BOOL;
		P3_Bunka_Zamky_AKTIVNE : BOOL;
		P3_ZonaBunky_AKTIVNA : BOOL;
		P3_ZonaHVtest_AKTIVNA : BOOL;
		P4_Panel_TlacitkoCS_ODBLOK : BOOL;
		P4_Rozvadzac_TlacitkoCS_ODBLOK : BOOL;
		P4_VyblokovanieZamkov_AKTIVNE : BOOL;
		P4_DeadMan_AKTIVNY : BOOL;
		P4_ZonaVytahu_AKTIVNA : BOOL;
		P4_Bunka_VstupBariera_AKTIVNA : BOOL;
		P4_ZonaBunky_AKTIVNA : BOOL;
		P4_Vytah_Bariera_AKTIVNA : BOOL;
		P4_Vytah_Muting_AKTIVNY : BOOL;
		P4_Bunka_Zamky_AKTIVNE : BOOL;
		P4_VystupBunky_VstupBar_AKTIVNA : BOOL;
		P4_VystupBunky_VystupBar_AKTIVNA : BOOL;
	END_STRUCT;
END_TYPE

(*************************************Linka všeobecne**********************************************)

TYPE
	Linka_typ : 	STRUCT
		IN : Linka_IN_typ;
		OUT : Linka_OUT_typ;
		PAR : Linka_PAR_typ;
		STAV : Linka_STAV_typ;
		Automat : BOOL;
		Manual : BOOL;
		Reset : BOOL;
		KoniecCyklu : BOOL;
		ZberFotiek : BOOL;
		KOM_Panatrace_OFF : BOOL;
		KOM_FTP_OFF : BOOL;
		P1_Kamery_OFF : BOOL;
		P2_Kamery_OFF : BOOL;
		P3_Kamery_OFF : BOOL;
		P4_Kamery_OFF : BOOL;
		P1_SkrutkovanieResult_OFF : BOOL;
		P2_SkrutkovanieResult_OFF : BOOL;
		P3_SkrutkovanieResult_OFF : BOOL;
	END_STRUCT;
	Linka_IN_typ : 	STRUCT
		SafetyMaster_OK : BOOL;
	END_STRUCT;
	Linka_OUT_typ : 	STRUCT
		New_Member : USINT;
	END_STRUCT;
	Linka_PAR_typ : 	STRUCT
		ZvolenyModel : STRING[2]; (*4F, 5F, 5H*)
		TestovaciKus : BOOL;
		RevorkovyKus : BOOL;
		PaletkaPrechadza : BOOL;
		IndexModelu : USINT;
		VyprazdnenieLinky : BOOL;
	END_STRUCT;
	Linka_STAV_typ : 	STRUCT
		PoINIT : BOOL;
		VyprazdnenieLinky : BOOL;
		OFF : BOOL;
		PRAZDNA : BOOL;
	END_STRUCT;
END_TYPE

(*************************************Pracovisko P1**************************************************)

TYPE
	P1_Pracovisko_typ : 	STRUCT
		IN : P1_Pracovisko_IN_typ;
		OUT : P1_Pracovisko_OUT_typ;
		PAR : P1_Pracovisko_PAR_typ;
		STAV : P1_Pracovisko_STAV_typ;
		COM_Weidmuller : P1_COM_Weidmuller_typ;
		COM_Festo : P1_COM_Festo_typ;
		COM_VentilovyTerminal : ARRAY[0..5]OF USINT;
		Automat : BOOL;
		Manual : BOOL;
		Reset : BOOL;
		KoniecCyklu : BOOL;
	END_STRUCT;
	P1_Pracovisko_IN_typ : 	STRUCT
		TlakVzduchu_OK : BOOL; (*S1_5*)
		ModulWeidmuller_IO_KomOK : BOOL;
		VentilovyTerminal_KomOK : BOOL;
		Robot_KomOK : BOOL;
		Skrutkovacka_K30_KomOK : BOOL;
		Skrutkovacka_M5_KomOK : BOOL;
		Skrutkovacka_M4_KomOK : BOOL;
		ModulFesto_IO_KomOK : BOOL;
		SmartKamera3_KomOK : BOOL;
		SmartKamera5_KomOK : BOOL;
		ServoZdvihuVytahu_KomOK : BOOL;
		ServoManipulatorOsX_KomOK : BOOL;
		ServoManipulatorOsY_KomOK : BOOL;
		ServoManipulatorOsZ_M5_KomOK : BOOL;
		ServoManipulatorOsZ_M4_KomOK : BOOL;
		PredneDvere_PritomnostAdaptera : BOOL; (*EZ 1.1*)
		ZadneDvere_PritomnostAdaptera : BOOL; (*EZ 1.2*)
	END_STRUCT;
	P1_Pracovisko_OUT_typ : 	STRUCT
		Majak_ZeleneSvetlo_ON : BOOL;
		Majak_OranzoveSvetlo_ON : BOOL;
		Majak_CerveneSvetlo_ON : BOOL;
		Majak_Hukacka_ON : BOOL;
		OsvetlenieBunky_ON : BOOL;
		Srobovanie_BodoveOsvetlenie_ON : BOOL;
		Srobovanie_OsvetleniePaletky_ON : BOOL;
		Osvetlenie_CAM4_ON : BOOL;
		Osvetlenie_CAM6_ON : BOOL;
		Osvetlenie_CAM5_ON : BOOL;
		PredneDvere_ZAMKNI : BOOL; (*EZ 1.1*)
		ZadneDvere_ZAMKNI : BOOL; (*EZ 1.2*)
	END_STRUCT;
	P1_Pracovisko_PAR_typ : 	STRUCT
		New_Member : USINT;
	END_STRUCT;
	P1_Pracovisko_STAV_typ : 	STRUCT
		Automat : BOOL;
		Manual : BOOL;
		PoINIT : BOOL;
		READY : BOOL;
		PORUCHA : BOOL;
		HardwareVytahu_OK : BOOL;
		HardwareBunky_OK : BOOL;
		SkrutkovackyZasunute : BOOL;
		Porucha_ST1 : BOOL; (*Vstupný výťah*)
		Porucha_ST2 : BOOL; (*Šrobovanie*)
		Porucha_ST3 : BOOL; (*Akumulačný stoper*)
		UkoncenieCyklu_BUSY : BOOL;
	END_STRUCT;
	P1_COM_Weidmuller_typ : 	STRUCT
		AB1_2_8DI : USINT;
		AB1_3_8DI : USINT;
		AB1_4_8DI : USINT;
		AB1_5_8DI : USINT;
		AB1_6_8DO : USINT;
		AB1_7_8DO : USINT;
		AB1_9_8DO : USINT;
		AB1_10_8DO : USINT;
	END_STRUCT;
	P1_COM_Festo_typ : 	STRUCT
		DM1_1_4DI : ARRAY[0..3]OF BOOL;
		DM1_1_4DO : ARRAY[0..3]OF BOOL;
		DI1_1_8DI : ARRAY[0..7]OF BOOL;
		DI1_2_8DI : ARRAY[0..7]OF BOOL;
		DI1_3_8DI : ARRAY[0..7]OF BOOL;
		DI1_4_8DI : ARRAY[0..7]OF BOOL;
		DI1_5_8DI : ARRAY[0..7]OF BOOL;
		DS1_1_Port0_IN : ARRAY[0..1]OF USINT;
		DS1_1_Port0_OUT : ARRAY[0..1]OF USINT;
		DS1_1_Port1_IN : ARRAY[0..15]OF USINT;
		DS1_1_Port1_OUT : ARRAY[0..15]OF USINT;
		DS1_1_Port2_IN : ARRAY[0..31]OF USINT;
		DS1_1_Port2_OUT : ARRAY[0..31]OF USINT;
		DS1_1_Port3_IN : ARRAY[0..31]OF USINT;
		DS1_1_Port3_OUT : ARRAY[0..31]OF USINT;
		DS1_2_Port0_IN : ARRAY[0..1]OF USINT;
		DS1_2_Port0_OUT : ARRAY[0..1]OF USINT;
	END_STRUCT;
END_TYPE

(*//P1 - Výťah//*)

TYPE
	P1_Vytah_typ : 	STRUCT
		CMD : P1_Vytah_CMD_typ;
		IN : P1_Vytah_IN_typ;
		OUT : P1_Vytah_OUT_typ;
		PAR : P1_Vytah_PAR_typ;
		STAV : P1_Vytah_STAV_typ;
		Banner : BannerIOlink;
		RFID_hlava : SickHeads; (*S_1.3*)
		ServoZdvihuVytahu : ServoDriver; (*M_1.1*)
		Automat : BOOL;
		Manual : BOOL;
		Reset : BOOL;
		KoniecCyklu : BOOL;
	END_STRUCT;
	P1_Vytah_CMD_typ : 	STRUCT
		RR_ChodDopravnika_VPRED : BOOL;
		RR_ChodDopravnika_VZAD : BOOL;
		RR_ZdvihVytahu_HORE : BOOL;
		RR_ZdvihVytahu_DOLE : BOOL;
		Banner_LED_OFF : BOOL;
	END_STRUCT;
	P1_Vytah_IN_typ : 	STRUCT
		PrechodDopravnika : BOOL; (*OS1_8*)
		Zdvih_HornyLimSnimac : BOOL; (*IS1_17*)
		Zdvih_SpodnyLimSnimac : BOOL; (*IS1_16*)
		StavRiadeniaDopravVytahu_READY : BOOL; (*M1_11*)
		TeplotaMotoraDopravVytahu_OK : BOOL; (*M1_11*)
	END_STRUCT;
	P1_Vytah_OUT_typ : 	STRUCT
		DopravnikChod_VPRED : BOOL; (*M1_11*)
		DopravnikChod_VZAD : BOOL; (*M1_11*)
		OsvetlenieVytahu_ON : BOOL;
	END_STRUCT;
	P1_Vytah_PAR_typ : 	STRUCT
		CisloPaletky_STRING : STRING[2];
		CisloPaletky : USINT;
		IndexFotky : USINT;
		StaryQRkod_PowerCP : STRING[30];
		StaryQRkod_DPS_4F5F : STRING[32];
		Zdvih_JoggRychlost : REAL;
		RR_PrecitaneCisloPaletky : USINT;
	END_STRUCT;
	P1_Vytah_STAV_typ : 	STRUCT
		PrebiehaVyvezeniePaletky : BOOL;
		PoINIT : BOOL;
	END_STRUCT;
END_TYPE

(*//P1 - Spodný stoper//*)

TYPE
	P1_SpodnyStoper_typ : 	STRUCT
		IN : P1_SpodnyStoper_IN_typ;
		OUT : P1_SpodnyStoper_OUT_typ;
		PAR : P1_SpodnyStoper_PAR_typ;
		STAV : P1_SpodnyStoper_STAV_typ;
		Automat : BOOL;
		Manual : BOOL;
		Reset : BOOL;
		KoniecCyklu : BOOL;
	END_STRUCT;
	P1_SpodnyStoper_IN_typ : 	STRUCT
		PritomnostPaletky : BOOL; (*IS1_4*)
		ZaplnenieDopravnika : BOOL; (*IS1_22*)
	END_STRUCT;
	P1_SpodnyStoper_OUT_typ : 	STRUCT
		ZasunStoper : BOOL; (*YV005_VT1*)
	END_STRUCT;
	P1_SpodnyStoper_PAR_typ : 	STRUCT
		New_Member : USINT;
	END_STRUCT;
	P1_SpodnyStoper_STAV_typ : 	STRUCT
		PoINIT : BOOL;
		PrebiehaVyvezeniePaletky : BOOL;
	END_STRUCT;
END_TYPE

(*//P1 - Dopravníky//*)

TYPE
	P1_Dopravniky_typ : 	STRUCT
		IN : P1_Dopravniky_IN_typ;
		OUT : P1_Dopravniky_OUT_typ;
		PAR : P1_Dopravniky_PAR_typ;
		STAV : P1_Dopravniky_STAV_typ;
		Automat : BOOL;
		Manual : BOOL;
		Reset : BOOL;
		KoniecCyklu : BOOL;
	END_STRUCT;
	P1_Dopravniky_IN_typ : 	STRUCT
		StavRiadeniaVratnehoDoprav_READY : BOOL; (*M1_13*)
		StavRiadeniaDopravBunky_READY : BOOL; (*M1_12*)
		TeplotaMotoraVratnehoDoprav_OK : BOOL; (*M1_13*)
		TeplotaMotoraDopravBunky_OK : BOOL; (*M1_12*)
	END_STRUCT;
	P1_Dopravniky_OUT_typ : 	STRUCT
		DopravnikBunky_ON : BOOL; (*M1_12*)
		VratnyDopravnik_ON : BOOL; (*M1_13*)
	END_STRUCT;
	P1_Dopravniky_PAR_typ : 	STRUCT
		New_Member : USINT;
	END_STRUCT;
	P1_Dopravniky_STAV_typ : 	STRUCT
		PoINIT : BOOL;
	END_STRUCT;
END_TYPE

(*//P1 - Stoper šrobovania//*)

TYPE
	P1_StoperSrobovania_typ : 	STRUCT
		CMD : P1_StoperSrobovania_CMD_typ;
		IN : P1_StoperSrobovania_IN_typ;
		OUT : P1_StoperSrobovania_OUT_typ;
		PAR : P1_StoperSrobovania_PAR_typ;
		STAV : P1_StoperSrobovania_STAV_typ;
		RFID_hlava : SickHeads;
		Automat : BOOL;
		Manual : BOOL;
		Reset : BOOL;
		KoniecCyklu : BOOL;
	END_STRUCT;
	P1_StoperSrobovania_CMD_typ : 	STRUCT
		RR_VysunCentrovanie : BOOL;
	END_STRUCT;
	P1_StoperSrobovania_IN_typ : 	STRUCT
		Centrovanie_VYSUNUTE : BOOL; (*IS1_1*)
		Centrovanie_ZASUNUTE : BOOL; (*IS1_2*)
	END_STRUCT;
	P1_StoperSrobovania_OUT_typ : 	STRUCT
		ZasunStoper : BOOL; (*YV001_VT1*)
		Centrovanie_VYSUN : BOOL; (*YV002_VT1*)
		Centrovanie_ZASUN : BOOL; (*YV003_VT1*)
	END_STRUCT;
	P1_StoperSrobovania_PAR_typ : 	STRUCT
		CisloPaletky_STRING : STRING[2];
		IndexFotky : USINT;
		CisloPaletky : USINT;
	END_STRUCT;
	P1_StoperSrobovania_STAV_typ : 	STRUCT
		PoINIT : BOOL;
		PrebiehaVyvezeniePaletky : BOOL;
		VstupnaKamerovaKontrola : BOOL;
		VyrobaZacala : BOOL;
	END_STRUCT;
END_TYPE

(*//P1 - Šrobovanie//*)

TYPE
	P1_Srobovanie_typ : 	STRUCT
		CMD : P1_Srobovanie_CMD_typ;
		IN : P1_Srobovanie_IN_typ;
		OUT : P1_Srobovanie_OUT_typ;
		PAR : P1_Srobovanie_PAR_typ;
		STAV : P1_Srobovanie_STAV_typ;
		COM_IN : P1_Srobovanie_COM_IN_typ;
		COM_OUT : P1_Srobovanie_COM_OUT_typ;
		Automat : BOOL;
		Manual : BOOL;
		Reset : BOOL;
		KoniecCyklu : BOOL;
		ServoManipulOsX : ServoDriver; (*M1_2*)
		ServoManipulOsY : ServoDriver; (*M1_3*)
		ServoManipulOsZ_M4 : ServoDriver; (*M1_5*)
		ServoManipulOsZ_M5 : ServoDriver; (*M1_4*)
		Skrutkovacka_K30 : SkrutkovackaAtlasCopco_typ;
		Skrutkovacka_M4 : SkrutkovackaAtlasCopco_typ;
		Skrutkovacka_M5 : SkrutkovackaAtlasCopco_typ;
		SkrutSet_K30 : ScrewLoading;
		SkrutSet_M5 : PickAndPlace;
		SkrutSet_M4 : PickAndPlace;
	END_STRUCT;
	P1_Srobovanie_CMD_typ : 	STRUCT
		RR_Manipulator_OsX_VPRAVO : BOOL;
		RR_Manipulator_OsX_VLAVO : BOOL;
		RR_Manipulator_OsY_VPRED : BOOL;
		RR_Manipulator_OsY_VZAD : BOOL;
		RR_SkrutkovackaM4_OsZ_HORE : BOOL;
		RR_SkrutkovackaM4_OsZ_DOLE : BOOL;
		RR_SkrutkovackaM5_OsZ_HORE : BOOL;
		RR_SkrutkovackaM5_OsZ_DOLE : BOOL;
		RR_PrisavanieSkrutkyM5_ON : BOOL;
		RR_PrisavanieSkrutkyM5_OFF : BOOL;
		RR_PrisavanieSkrutkyM4_ON : BOOL;
		RR_PrisavanieSkrutkyM4_OFF : BOOL;
		RR_CistenieSkrutkovackyK30 : BOOL;
		RR_SkrutSetK30_Zasobnik_RUN : BOOL;
		RR_SkrutSetK30_PodajSkrutku : BOOL;
		RR_SkrutSetK30_VysunBrzdu : BOOL;
		RR_SkrutSetM4_Zasobnik_RUN : BOOL;
		RR_SkrutSetM4_Vibrolista_RUN : BOOL;
		RR_SkrutSetM4_PodajSkrutku : BOOL;
		RR_SkrutSetM4_OtocPodavac_Vstup : BOOL;
		RR_SkrutSetM4_OtocPodavac_Vystup : BOOL;
		RR_SkrutSetM5_Zasobnik_RUN : BOOL;
		RR_SkrutSetM5_Vibrolista_RUN : BOOL;
		RR_SkrutSetM5_PodajSkrutku : BOOL;
		RR_SkrutSetM5_OtocPodavac_Vstup : BOOL;
		RR_SkrutSetM5_OtocPodavac_Vystup : BOOL;
		RR_PolohujManipulator : BOOL;
		PodajSkrutku_K30 : BOOL;
		PodajSkrutku_M4 : BOOL;
		PodajSkrutku_M5 : BOOL;
	END_STRUCT;
	P1_Srobovanie_IN_typ : 	STRUCT
		ManipulOsX_LimSnimac_POS : BOOL; (*IS1_21*)
		ManipulOsX_LimSnimac_NEG : BOOL; (*IS1_20*)
		ManipulOsY_LimSnimac_POS : BOOL; (*IS1_19*)
		ManipulOsY_LimSnimac_NEG : BOOL; (*IS1_18*)
		ManipulOsZ_M4_LimSnimacHorny : BOOL; (*IS1_24*)
		ManipulOsZ_M4_LimSnimacSpodny : BOOL; (*IS1_25*)
		ManipulOsZ_M5_LimSnimacHorny : BOOL; (*IS1_5*)
		ManipulOsZ_M5_LimSnimacSpodny : BOOL; (*IS1_6*)
		Skrutkovacka_K30_ZASUNUTA : BOOL; (*MS1_7*)
		Skrutkovacka_M5_Vakum_OK : BOOL; (*S1_6*)
		Skrutkovacka_M4_Vakum_OK : BOOL; (*S1_7*)
		NapajanieSkrutkovackyM4_OK : BOOL;
		NapajanieSkrutkovackyK30_OK : BOOL;
		NapajanieSkrutkovackyM5_OK : BOOL;
		NapajanieZasobnikaK30_OK : BOOL;
		NapajanieZasobnikaM5_OK : BOOL;
		NapajanieZasobnikaM4_OK : BOOL;
		NapajanieVibrolistyM5_OK : BOOL;
		NapajanieVibrolistyM4_OK : BOOL;
	END_STRUCT;
	P1_Srobovanie_OUT_typ : 	STRUCT
		Skrutkovacku_K30_VYSUN : BOOL; (*YV018_VT1*)
		Skrutkovacka_K30_Prisavanie_ON : BOOL; (*YV016_VT1*)
		Skrutkovacka_K30_Odvzdusn_ON : BOOL; (*YV017_VT1*)
		Skrutkovacka_M4_Prisavanie_ON : BOOL; (*YV025_VT1*)
		Skrutkovacka_M4_Prisavanie_OFF : BOOL; (*YV026_VT1*)
		Skrutkovacka_M4_Odvzdusn_ON : BOOL; (*YV027_VT1*)
		Skrutkovacka_M5_Prisavanie_ON : BOOL; (*YV022_VT1*)
		Skrutkovacka_M5_Prisavanie_OFF : BOOL; (*YV023_VT1*)
		Skrutkovacka_M5_Odvzdusn_ON : BOOL; (*YV024_VT1*)
	END_STRUCT;
	P1_Srobovanie_PAR_typ : 	STRUCT
		RR_IndexPolohovaniaManipulatora : USINT;
		RR_TypModelu : STRING[2];
		Skrutkov_K30_AktualHodnVysunutia : UINT; (*IO-Link snímač*)
		Skrutkov_K30_RoundHodnotaREAL : REAL;
		ManipulOsX_AktualnaPozicia : REAL;
		ManipulOsY_AktualnaPozicia : REAL;
		ManipulOsZ_M5_AktualnaPozicia : REAL;
		ManipulOsZ_M4_AktualnaPozicia : REAL;
		ManipulOsX_JoggRychlost : REAL;
		ManipulOsY_JoggRychlost : REAL;
		ManipulOsZ_M5_JoggRychlost : REAL;
		ManipulOsZ_M4_JoggRychlost : REAL;
		K30_AtlasCopcoInputs : ARRAY[0..7]OF UDINT;
		K30_AtlasCopcoOutputs : ARRAY[0..7]OF UDINT;
		M5_AtlasCopcoInputs : ARRAY[0..7]OF UDINT;
		M5_AtlasCopcoOutputs : ARRAY[0..7]OF UDINT;
		M4_AtlasCopcoInputs : ARRAY[0..7]OF UDINT;
		M4_AtlasCopcoOutputs : ARRAY[0..7]OF UDINT;
	END_STRUCT;
	P1_Srobovanie_STAV_typ : 	STRUCT
		RR_Polohovanie_BUSY : BOOL;
		PoINIT : BOOL;
		Vysledok_Srobovania : STRING[2]; (*OK alebo NG*)
		K30_DosiahnutyMoment_REAL : REAL;
		K30_DosiahnutyMoment : UDINT;
		K30_Moment_ToleranciaMAX_REAL : REAL;
		K30_Moment_ToleranciaMAX : UDINT;
		K30_Moment_ToleranciaMIN_REAL : REAL;
		K30_Moment_ToleranciaMIN : UDINT;
		K30_DosiahnutyUhol : UINT;
		K30_Uhol_ToleranciaMAX_REAL : REAL;
		K30_Uhol_ToleranciaMAX : UDINT;
		K30_Uhol_ToleranciaMIN_REAL : REAL;
		K30_Uhol_ToleranciaMIN : UDINT;
		M5_DosiahnutyMoment_REAL : REAL;
		M5_DosiahnutyMoment : UDINT;
		M5_Moment_ToleranciaMAX_REAL : REAL;
		M5_Moment_ToleranciaMAX : UDINT;
		M5_Moment_ToleranciaMIN_REAL : REAL;
		M5_Moment_ToleranciaMIN : UDINT;
		M5_DosiahnutyUhol : UINT;
		M5_Uhol_ToleranciaMAX_REAL : REAL;
		M5_Uhol_ToleranciaMAX : UDINT;
		M5_Uhol_ToleranciaMIN_REAL : REAL;
		M5_Uhol_ToleranciaMIN : UDINT;
		M4_DosiahnutyMoment_REAL : REAL;
		M4_DosiahnutyMoment : UDINT;
		M4_Moment_ToleranciaMAX_REAL : REAL;
		M4_Moment_ToleranciaMAX : UDINT;
		M4_Moment_ToleranciaMIN_REAL : REAL;
		M4_Moment_ToleranciaMIN : UDINT;
		M4_DosiahnutyUhol : UINT;
		M4_Uhol_ToleranciaMAX_REAL : REAL;
		M4_Uhol_ToleranciaMAX : UDINT;
		M4_Uhol_ToleranciaMIN_REAL : REAL;
		M4_Uhol_ToleranciaMIN : UDINT;
		ManipulatorNadPodavacmi : BOOL;
		SkrutkaK30_READY : BOOL;
		CistenieSkrutkovackyK30_BUSY : BOOL;
	END_STRUCT;
	P1_Srobovanie_COM_IN_typ : 	STRUCT
		PresunManipulatora_VPRED : BOOL;
		PresunManipulatora_VZAD : BOOL;
		OdoberSkrutku_M5 : BOOL;
		OdoberSkrutku_M4 : BOOL;
		Model45F_ZaskrutkujLavu_K30 : BOOL;
		Model45F_ZaskrutkujPravu_K30 : BOOL;
		Model5H_ZaskrutkujLavu_K30 : BOOL;
		Model5H_ZaskrutkujPravu_K30 : BOOL;
		Model45F_ZaskrutkujPrednu_M4 : BOOL;
		Model45F_ZaskrutkujZadnu_M4 : BOOL;
		Model45F_ZaskrutkujDPS_M4 : BOOL;
		Model5H_ZaskrutkujLavu_M5 : BOOL;
		Model5H_ZaskrutkujPravu_M5 : BOOL;
		Model5H_ZaskrutkujStrednu_M5 : BOOL;
	END_STRUCT;
	P1_Srobovanie_COM_OUT_typ : 	STRUCT
		Stav_SkrutkovanieUkoncene : BOOL;
		Stav_PresunManipulUkonceny : BOOL;
		Stav_PoruchaSkrutkovania : BOOL;
	END_STRUCT;
END_TYPE

(*//P1 - Akumulačný stoper//*)

TYPE
	P1_AkumulacnyStoper_typ : 	STRUCT
		IN : P1_AkumulacnyStoper_IN_typ;
		OUT : P1_AkumulacnyStoper_OUT_typ;
		PAR : P1_AkumulacnyStoper_PAR_typ;
		STAV : P1_AkumulacnyStoper_STAV_typ;
		Automat : BOOL;
		Manual : BOOL;
		Reset : BOOL;
		KoniecCyklu : BOOL;
	END_STRUCT;
	P1_AkumulacnyStoper_IN_typ : 	STRUCT
		PritomnostPaletky : BOOL; (*IS1_3*)
	END_STRUCT;
	P1_AkumulacnyStoper_OUT_typ : 	STRUCT
		ZasunStoper : BOOL; (*YV004_VT1*)
	END_STRUCT;
	P1_AkumulacnyStoper_PAR_typ : 	STRUCT
		New_Member : USINT;
	END_STRUCT;
	P1_AkumulacnyStoper_STAV_typ : 	STRUCT
		PoINIT : BOOL;
		PrebiehaVyvezeniePaletky : BOOL;
	END_STRUCT;
END_TYPE

(*//P1 - Robot//*)

TYPE
	P1_Robot_typ : 	STRUCT
		CMD : P1_Robot_CMD_typ;
		IN : P1_Robot_IN_typ;
		OUT : P1_Robot_OUT_typ;
		PAR : P1_Robot_PAR_typ;
		STAV : P1_Robot_STAV_typ;
		COM_IN : P1_Robot_COM_IN_typ;
		COM_OUT : P1_Robot_COM_OUT_typ;
		Automat : BOOL;
		Manual : BOOL;
		Reset : BOOL;
		KoniecCyklu : BOOL;
	END_STRUCT;
	P1_Robot_CMD_typ : 	STRUCT
		New_Member : USINT;
	END_STRUCT;
	P1_Robot_IN_typ : 	STRUCT
		Vakum_OK : BOOL; (*S1_4*)
		DokStanica_PritomnGripra45F : BOOL; (*IS1_23*)
		DokStanica_PritomnGripra5H : BOOL; (*IS1_13*)
		TypGripra_45F : BOOL;
		TypGripra_5H : BOOL;
		Griper45F_Otvoreny : BOOL; (*MS1_10*)
		Griper45F_Zatvoreny : BOOL; (*MS1_11*)
		KodGripra_Bit0 : BOOL;
		KodGripra_Bit1 : BOOL;
	END_STRUCT;
	P1_Robot_OUT_typ : 	STRUCT
		Griper_OTVOR : BOOL; (*YV008_VT1*)
		Griper_ZATVOR : BOOL; (*YV009_VT1*)
		OdistiGriper : BOOL; (*YV007_VT1*)
		ZaistiGriper : BOOL; (*YV006_VT1*)
		Vakum_ON : BOOL; (*YV010_VT1*)
		Vakum_OFF : BOOL; (*YV011_VT1*)
	END_STRUCT;
	P1_Robot_PAR_typ : 	STRUCT
		New_Member : USINT;
	END_STRUCT;
	P1_Robot_STAV_typ : 	STRUCT
		PoINIT : BOOL;
		DrziFoamy_45F : BOOL;
		DrziBusbar_45F : BOOL;
		DrziBusbar_5H : BOOL;
		DrziDPS_45F : BOOL;
	END_STRUCT;
	P1_Robot_COM_IN_typ : 	STRUCT
		BYTE_IN : ARRAY[0..63]OF USINT; (*Z robota do PLC*)
		Stav_RobotOdparkovany : BOOL;
		Stav_RobotPoziciaCakania : BOOL;
		Stav_RobotBezpPozicia_Srobovanie : BOOL;
		Stav_MotoryON : BOOL;
		Stav_MotoryOFF : BOOL;
		Stav_ProgramRUN : BOOL;
		Stav_RezimAUTOMAT : BOOL;
		Stav_RobotCS : BOOL;
		Stav_VystupyZresetovane : BOOL;
		Stav_Foam4F_Odobraty : BOOL;
		Stav_Foam5F_Odobraty : BOOL;
		Stav_Foam4F_Polozeny : BOOL;
		Stav_Foam5F_Polozeny : BOOL;
		Stav_SpodnyBusbar4F_Odobraty : BOOL;
		Stav_SpodnyBusbar5F_Odobraty : BOOL;
		Stav_SpodnyBusbar4F_Polozeny : BOOL;
		Stav_SpodnyBusbar5F_Polozeny : BOOL;
		Stav_DPS_4F_Odobraty : BOOL;
		Stav_DPS_5F_Odobraty : BOOL;
		Stav_DPS_4F_Polozeny : BOOL;
		Stav_DPS_5F_Polozeny : BOOL;
		Stav_SpodnyBusbar5H_Odobraty : BOOL;
		Stav_SpodnyBusbar5H_Polozeny : BOOL;
		Stav_BusbaryUvolnene : BOOL;
		Stav_RobotOdoberaBusbary : BOOL;
		Stav_RobotOdoberaFoamy : BOOL;
	END_STRUCT;
	P1_Robot_COM_OUT_typ : 	STRUCT
		BYTE_OUT : ARRAY[0..63]OF USINT; (*Z PLC do Robota*)
		ManipSrobovania_BezpecnaPozicia : BOOL;
		OdoberFoam4F_z_Paletky : BOOL;
		OdoberFoam5F_z_Paletky : BOOL;
		PolozFoam4F_na_PowerCP : BOOL;
		PolozFoam5F_na_PowerCP : BOOL;
		OdoberSpodnyBusbar4F_z_Paletky : BOOL;
		OdoberSpodnyBusbar5F_z_Paletky : BOOL;
		PolozSpodnyBusbar4F_na_PowerCP : BOOL;
		PolozSpodnyBusbar5F_na_PowerCP : BOOL;
		OdoberDPS_4F_z_Paletky : BOOL;
		OdoberDPS_5F_z_Paletky : BOOL;
		PolozDPS_4F_na_PowerCP : BOOL;
		PolozDPS_5F_na_PowerCP : BOOL;
		OdoberSpodnyBusbar5H_z_Paletky : BOOL;
		PolozSpodnyBusbar5H_na_PowerCP : BOOL;
		UvolniBusbary : BOOL;
		Presun_CakaciaPozicia : BOOL;
		Odparkovanie : BOOL;
		ZapniMotory : BOOL;
		VypniMotory : BOOL;
		PP_na_Main : BOOL;
		Reset_CS : BOOL;
		StartProgramu : BOOL;
		StartProgramuMain : BOOL;
		StopProgramu : BOOL;
		TypGripra_5H : BOOL;
		TypGripra_45F : BOOL;
		ZopakujOdoberanie : BOOL;
	END_STRUCT;
END_TYPE

(***********************************Pracovisko 2****************************************************************)

TYPE
	P2_Pracovisko_typ : 	STRUCT
		IN : P2_Pracovisko_IN_typ;
		OUT : P2_Pracovisko_OUT_typ;
		PAR : P2_Pracovisko_PAR_typ;
		STAV : P2_Pracovisko_STAV_typ;
		Automat : BOOL;
		Manual : BOOL;
		Reset : BOOL;
		KoniecCyklu : BOOL;
		COM_Weidmuller : P2_COM_Weidmuller_typ;
		COM_Festo : P2_COM_Festo_typ;
		COM_VentilovyTerminal : ARRAY[0..10]OF USINT;
	END_STRUCT;
	P2_Pracovisko_IN_typ : 	STRUCT
		TlakVzduchu_OK : BOOL; (*S2_10*)
		ModulWeidmuller_IO_KomOK : BOOL;
		VentilovyTerminal_KomOK : BOOL;
		Robot_KomOK : BOOL;
		Skrutkovacka_M6_KomOK : BOOL;
		Skrutkovacka_M5_KomOK : BOOL;
		Skrutkovacka_M4_KomOK : BOOL;
		Maticovacka_M4_KomOK : BOOL;
		ModulFesto_IO_KomOK : BOOL;
		SafetyModul_KomOK : BOOL;
		SmartKamera8_KomOK : BOOL;
		SmartKamera9_KomOK : BOOL;
		ServoManipulatorOsX_KomOK : BOOL;
		ServoManipulatorOsY_KomOK : BOOL;
		ServoManipulatorOsZ_M4_KomOK : BOOL;
		ServoZaklTesneniaPojazd_KomOK : BOOL;
		ServoZaklTesneniaZdvih_KomOK : BOOL;
		ServoZvaraniaOsZ_KomOK : BOOL;
		PredneDvereLS_PritomnostAdaptera : BOOL;
		PredneDverePS_PritomnostAdaptera : BOOL;
		ZadneDvereLS_PritomnostAdaptera : BOOL;
		ZadneDverePS_PritomnostAdaptera : BOOL;
	END_STRUCT;
	P2_Pracovisko_OUT_typ : 	STRUCT
		Majak_ZeleneSvetlo_ON : BOOL;
		Majak_OranzoveSvetlo_ON : BOOL;
		Majak_CerveneSvetlo_ON : BOOL;
		Majak_Hukacka_ON : BOOL;
		OsvetlenieBunky_ON : BOOL;
		OsvetleniePracZaklTesnenia_ON : BOOL;
		Osvetlenie_CAM1_Svetlo1 : BOOL; (*Zakladač tesnenia*)
		Osvetlenie_CAM1_Svetlo2 : BOOL; (*Zakladač tesnenia*)
		Osvetlenie_CAM10 : BOOL; (*Stoper skrutkovania matic*)
		Osvetlenie_CAM11 : BOOL; (*Stoper zvárania*)
		Osvetlenie_CAM12 : BOOL; (*Stoper srobovania*)
		Srobovanie_BodoveOsvetlenie_ON : BOOL;
		Srobovanie_OsvetleniePaletky_ON : BOOL;
		PredneDvereLS_ZAMKNI : BOOL;
		PredneDverePS_ZAMKNI : BOOL;
		ZadneDvereLS_ZAMKNI : BOOL;
		ZadneDverePS_ZAMKNI : BOOL;
	END_STRUCT;
	P2_Pracovisko_PAR_typ : 	STRUCT
		New_Member : USINT;
	END_STRUCT;
	P2_Pracovisko_STAV_typ : 	STRUCT
		Automat : BOOL;
		Manual : BOOL;
		PoINIT : BOOL;
		READY : BOOL;
		PORUCHA : BOOL;
		Porucha_ST1 : BOOL; (*Zakladanie tesnenia*)
		Porucha_ST2 : BOOL; (*Skrutkovanie matice*)
		Porucha_ST3 : BOOL; (*Akumulačný stoper*)
		Porucha_ST4 : BOOL; (*Šrobovanie*)
		Porucha_ST5 : BOOL; (*Zvaranie,Čistenie*)
		HardwareBunky_OK : BOOL;
		HardwareZaklTesnenia_OK : BOOL;
		SkrutkovackyZasunute : BOOL;
		UkoncenieCyklu_BUSY : BOOL;
		PredneDvereZamknute : BOOL;
		ZadneDvereZamknute : BOOL;
	END_STRUCT;
	P2_COM_Weidmuller_typ : 	STRUCT
		AB2_5_8DI : USINT;
		AB2_6_8DI : USINT;
		AB2_7_8DI : USINT;
		AB2_8_8DI : USINT;
		AB2_9_8DO : USINT;
		AB2_10_8DO : USINT;
		AB2_12_8DO : USINT;
		AB2_13_8DO : USINT;
	END_STRUCT;
	P2_COM_Festo_typ : 	STRUCT
		DI2_1_8DI : ARRAY[0..7]OF BOOL;
		DI2_2_8DI : ARRAY[0..7]OF BOOL;
		DI2_3_8DI : ARRAY[0..7]OF BOOL;
		DI2_4_8DI : ARRAY[0..7]OF BOOL;
		DI2_5_8DI : ARRAY[0..7]OF BOOL;
		DI2_6_8DI : ARRAY[0..7]OF BOOL;
		DI2_7_8DI : ARRAY[0..7]OF BOOL;
		DI2_8_8DI : ARRAY[0..7]OF BOOL;
		DM2_1_4DI : ARRAY[0..3]OF BOOL;
		DM2_1_4DO : ARRAY[0..3]OF BOOL;
		DS2_1_Port0_IN : ARRAY[0..1]OF USINT;
		DS2_1_Port0_OUT : ARRAY[0..1]OF USINT;
		DS2_1_Port1_IN : ARRAY[0..1]OF USINT;
		DS2_1_Port1_OUT : ARRAY[0..1]OF USINT;
		DS2_1_Port2_IN : ARRAY[0..1]OF USINT;
		DS2_1_Port2_OUT : ARRAY[0..1]OF USINT;
		DS2_1_Port3_IN : ARRAY[0..31]OF USINT;
		DS2_1_Port3_OUT : ARRAY[0..31]OF USINT;
		DS2_2_Port0_IN : ARRAY[0..31]OF USINT;
		DS2_2_Port0_OUT : ARRAY[0..31]OF USINT;
		DS2_2_Port1_IN : ARRAY[0..31]OF USINT;
		DS2_2_Port1_OUT : ARRAY[0..31]OF USINT;
		DS2_2_Port2_IN : ARRAY[0..31]OF USINT;
		DS2_2_Port2_OUT : ARRAY[0..31]OF USINT;
		DS2_2_Port3_IN : ARRAY[0..31]OF USINT;
		DS2_2_Port3_OUT : ARRAY[0..31]OF USINT;
		DS2_3_Port0_IN : ARRAY[0..15]OF USINT;
		DS2_3_Port0_OUT : ARRAY[0..15]OF USINT;
		DS2_3_Port1_IN : ARRAY[0..1]OF USINT;
		DS2_3_Port1_OUT : ARRAY[0..1]OF USINT;
	END_STRUCT;
END_TYPE

(*//P2 - Dopravníky//*)

TYPE
	P2_Dopravniky_typ : 	STRUCT
		IN : P2_Dopravniky_IN_typ;
		OUT : P2_Dopravniky_OUT_typ;
		PAR : P2_Dopravniky_PAR_typ;
		STAV : P2_Dopravniky_STAV_typ;
		Automat : BOOL;
		Manual : BOOL;
		Reset : BOOL;
		KoniecCyklu : BOOL;
	END_STRUCT;
	P2_Dopravniky_IN_typ : 	STRUCT
		StavRiadeniaVratnehoDoprav_READY : BOOL; (*M2_13*)
		StavRiadeniaDopravBunky_READY : BOOL; (*M2_12*)
		TeplotaMotoraVratnehoDoprav_OK : BOOL; (*M2_13*)
		TeplotaMotoraDopravBunky_OK : BOOL; (*M2_12*)
	END_STRUCT;
	P2_Dopravniky_OUT_typ : 	STRUCT
		DopravnikBunky_ON : BOOL; (*M2_12*)
		VratnyDopravnik_ON : BOOL; (*M2_13*)
	END_STRUCT;
	P2_Dopravniky_PAR_typ : 	STRUCT
		New_Member : USINT;
	END_STRUCT;
	P2_Dopravniky_STAV_typ : 	STRUCT
		PoINIT : BOOL;
	END_STRUCT;
END_TYPE

(*//P2 - Spodný stoper//*)

TYPE
	P2_SpodnyStoper_typ : 	STRUCT
		IN : P2_SpodnyStoper_IN_typ;
		OUT : P2_SpodnyStoper_OUT_typ;
		PAR : P2_SpodnyStoper_PAR_typ;
		STAV : P2_SpodnyStoper_STAV_typ;
		Automat : BOOL;
		Manual : BOOL;
		Reset : BOOL;
		KoniecCyklu : BOOL;
	END_STRUCT;
	P2_SpodnyStoper_IN_typ : 	STRUCT
		PritomnostPaletky : BOOL; (*IS2_8*)
		ZaplnenieDopravnika : BOOL; (*IS2_9*)
	END_STRUCT;
	P2_SpodnyStoper_OUT_typ : 	STRUCT
		ZasunStoper : BOOL; (*YV048_VT2*)
	END_STRUCT;
	P2_SpodnyStoper_PAR_typ : 	STRUCT
		New_Member : USINT;
	END_STRUCT;
	P2_SpodnyStoper_STAV_typ : 	STRUCT
		PoINIT : BOOL;
		PrebiehaVyvezeniePaletky : BOOL;
	END_STRUCT;
END_TYPE

(*//P2 - Stoper zakladaca tesnenia//*)

TYPE
	P2_StoperZaklTesnenia_typ : 	STRUCT
		CMD : P2_StoperZaklTesnenia_CMD_typ;
		IN : P2_StoperZaklTesnenia_IN_typ;
		OUT : P2_StoperZaklTesnenia_OUT_typ;
		PAR : P2_StoperZaklTesnenia_PAR_typ;
		STAV : P2_StoperZaklTesnenia_STAV_typ;
		Banner : BannerIOlink;
		RFID_hlava : SickHeads;
		Automat : BOOL;
		Manual : BOOL;
		Reset : BOOL;
		KoniecCyklu : BOOL;
	END_STRUCT;
	P2_StoperZaklTesnenia_CMD_typ : 	STRUCT
		Banner_LED_OFF : BOOL;
	END_STRUCT;
	P2_StoperZaklTesnenia_IN_typ : 	STRUCT
		New_Member : USINT;
	END_STRUCT;
	P2_StoperZaklTesnenia_OUT_typ : 	STRUCT
		ZasunStoper : BOOL; (*YV037_VT2*)
	END_STRUCT;
	P2_StoperZaklTesnenia_PAR_typ : 	STRUCT
		CisloPaletky_STRING : STRING[2];
		IndexFotky : USINT;
		StaryQRkod_Filtra5H : STRING[32];
		CisloPaletky : USINT;
	END_STRUCT;
	P2_StoperZaklTesnenia_STAV_typ : 	STRUCT
		PoINIT : BOOL;
		PrebiehaVyvezeniePaletky : BOOL;
		ObsluhaOznacilaPaletku_NG : BOOL;
	END_STRUCT;
END_TYPE

(*//P2 - Zakladač tesnenia//*)

TYPE
	P2_ZakladacTesnenia_typ : 	STRUCT
		CMD : P2_ZakladacTesnenia_CMD_typ;
		IN : P2_ZakladacTesnenia_IN_typ;
		OUT : P2_ZakladacTesnenia_OUT_typ;
		PAR : P2_ZakladacTesnenia_PAR_typ;
		STAV : P2_ZakladacTesnenia_STAV_typ;
		COM_IN : P2_ZakladacTesnenia_COM_IN_typ;
		COM_OUT : P2_ZakladacTesnenia_COM_OUT_typ;
		Automat : BOOL;
		Manual : BOOL;
		Reset : BOOL;
		KoniecCyklu : BOOL;
		ServoZdvihuZakladaca : ServoDriver;
		ServoPojazduZakladaca : ServoDriver;
	END_STRUCT;
	P2_ZakladacTesnenia_CMD_typ : 	STRUCT
		RR_PojazdZakladaca_VYSUN : BOOL;
		RR_PojazdZakladaca_ZASUN : BOOL;
		RR_ZdvihZakladaca_HORE : BOOL;
		RR_ZdvihZakladaca_DOLE : BOOL;
	END_STRUCT;
	P2_ZakladacTesnenia_IN_typ : 	STRUCT
		ZdvihZakladaca_HornyLimSnimac : BOOL; (*IS2_35*)
		Kopito_ZakladPoloha : BOOL; (*IS2_34*)
		Pojazd_PritomPowerCP : BOOL; (*OS2_4*)
	END_STRUCT;
	P2_ZakladacTesnenia_OUT_typ : 	STRUCT
		LED_DvojrucneOvladanie_ON : BOOL;
	END_STRUCT;
	P2_ZakladacTesnenia_PAR_typ : 	STRUCT
		IndexPaletky : USINT;
		ZakladacPojazd_JoggRychlost : REAL;
		ZakladacZdvih_JoggRychlost : REAL;
	END_STRUCT;
	P2_ZakladacTesnenia_STAV_typ : 	STRUCT
		PoINIT : BOOL;
	END_STRUCT;
	P2_ZakladacTesnenia_COM_IN_typ : 	STRUCT
		ZalozTesnenie : BOOL;
	END_STRUCT;
	P2_ZakladacTesnenia_COM_OUT_typ : 	STRUCT
		Stav_ZalozenieTesneniaUkoncene : BOOL;
		VysledokZalozeniaTesnenia : STRING[2]; (*OK alebo NG*)
	END_STRUCT;
END_TYPE

(*//P2 - Stoper matícovačky//*)

TYPE
	P2_StoperMaticovacky_typ : 	STRUCT
		CMD : P2_StoperMaticovacky_CMD_typ;
		IN : P2_StoperMaticovacky_IN_typ;
		OUT : P2_StoperMaticovacky_OUT_typ;
		PAR : P2_StoperMaticovacky_PAR_typ;
		STAV : P2_StoperMaticovacky_STAV_typ;
		Automat : BOOL;
		Manual : BOOL;
		Reset : BOOL;
		KoniecCyklu : BOOL;
		RFID_hlava : SickHeads;
		Maticovacka_M4 : SkrutkovackaAtlasCopco_typ;
		SkrutSet_MaticaM4 : MaticaSet;
	END_STRUCT;
	P2_StoperMaticovacky_CMD_typ : 	STRUCT
		RR_VysunCentrovanie : BOOL;
	END_STRUCT;
	P2_StoperMaticovacky_IN_typ : 	STRUCT
		Centrovanie_VYSUNUTE : BOOL; (*IS2_1*)
		Centrovanie_ZASUNUTE : BOOL; (*IS2_2*)
		Maticovacka_M4_ZASUNUTA : BOOL; (*MS2_5*)
	END_STRUCT;
	P2_StoperMaticovacky_OUT_typ : 	STRUCT
		ZasunStoper : BOOL; (*YV038_VT2*)
		Centrovanie_VYSUN : BOOL; (*YV039_VT2*)
		Centrovanie_ZASUN : BOOL; (*VY040_VT2*)
		Maticovacku_M4_VYSUN : BOOL; (*YV072_VT2*)
		Maticovacka_M4_Pneuzamok_ODOMKNI : BOOL; (*YV074_VT2*)
		Maticovacka_M4_Prisavanie_ON : BOOL; (*YV070_VT2*)
		Maticovacka_M4_Odvzdusn_ON : BOOL; (*YV071_VT2*)
	END_STRUCT;
	P2_StoperMaticovacky_PAR_typ : 	STRUCT
		CisloPaletky_STRING : STRING[2];
		IndexFotky : USINT;
		Maticov_M4_AktualHodnVysunutia : UINT; (*IO-Link snímač*)
		Maticov_M4_RoundHodnotaREAL : REAL;
		MaticeM4_AtlasCopcoInputs : ARRAY[0..7]OF UDINT;
		MaticeM4_AtlasCopcoOutputs : ARRAY[0..7]OF UDINT;
		CisloPaletky : USINT;
	END_STRUCT;
	P2_StoperMaticovacky_STAV_typ : 	STRUCT
		PoINIT : BOOL;
		PrebiehaVyvezeniePaletky : BOOL;
		VysledokSkrutkovaniaMatice : STRING[2]; (*OK alebo NG*)
		DosiahnutyMoment_REAL : REAL;
		DosiahnutyMoment : UDINT;
		Moment_ToleranciaMAX_REAL : REAL;
		Moment_ToleranciaMAX : UDINT;
		Moment_ToleranciaMIN_REAL : REAL;
		Moment_ToleranciaMIN : UDINT;
		DosiahnutyUhol : UINT;
		Uhol_ToleranciaMAX_REAL : REAL;
		Uhol_ToleranciaMAX : UDINT;
		Uhol_ToleranciaMIN_REAL : REAL;
		Uhol_ToleranciaMIN : UDINT;
		VstupnaKamerovaKontrola : BOOL;
		VyrobaZacala : BOOL;
	END_STRUCT;
END_TYPE

(*//P2 - Akumulačný stoper//*)

TYPE
	P2_AkumulacnyStoper_typ : 	STRUCT
		IN : P2_AkumulacnyStoper_IN_typ;
		OUT : P2_AkumulacnyStoper_OUT_typ;
		PAR : P2_AkumulacnyStoper_PAR_typ;
		STAV : P2_AkumulacnyStoper_STAV_typ;
		Automat : BOOL;
		Manual : BOOL;
		Reset : BOOL;
		KoniecCyklu : BOOL;
	END_STRUCT;
	P2_AkumulacnyStoper_IN_typ : 	STRUCT
		PritomnostPaletky : BOOL; (*IS2_3*)
	END_STRUCT;
	P2_AkumulacnyStoper_OUT_typ : 	STRUCT
		ZasunStoper : BOOL; (*YV041_VT2*)
	END_STRUCT;
	P2_AkumulacnyStoper_PAR_typ : 	STRUCT
		New_Member : USINT;
	END_STRUCT;
	P2_AkumulacnyStoper_STAV_typ : 	STRUCT
		PoINIT : BOOL;
		PrebiehaVyvezeniePaletky : BOOL;
	END_STRUCT;
END_TYPE

(*//P2 - Stoper šrobovania//*)

TYPE
	P2_StoperSrobovania_typ : 	STRUCT
		CMD : P2_StoperSrobovania_CMD_typ;
		IN : P2_StoperSrobovania_IN_typ;
		OUT : P2_StoperSrobovania_OUT_typ;
		PAR : P2_StoperSrobovania_PAR_typ;
		STAV : P2_StoperSrobovania_STAV_typ;
		RFID_hlava : SickHeads;
		Automat : BOOL;
		Manual : BOOL;
		Reset : BOOL;
		KoniecCyklu : BOOL;
	END_STRUCT;
	P2_StoperSrobovania_CMD_typ : 	STRUCT
		RR_VysunCentrovanie : BOOL;
	END_STRUCT;
	P2_StoperSrobovania_IN_typ : 	STRUCT
		Centrovanie_VYSUNUTE : BOOL; (*IS2_4*)
		Centrovanie_ZASUNUTE : BOOL; (*IS2_5*)
	END_STRUCT;
	P2_StoperSrobovania_OUT_typ : 	STRUCT
		ZasunStoper : BOOL; (*YV042_VT2*)
		Centrovanie_VYSUN : BOOL; (*YV043_VT2*)
		Centrovanie_ZASUN : BOOL; (*YV044_VT2*)
	END_STRUCT;
	P2_StoperSrobovania_PAR_typ : 	STRUCT
		CisloPaletky_STRING : STRING[2];
		IndexFotky : USINT;
		CisloPaletky : USINT;
	END_STRUCT;
	P2_StoperSrobovania_STAV_typ : 	STRUCT
		PoINIT : BOOL;
		PrebiehaVyvezeniePaletky : BOOL;
		VstupnaKamerovaKontrola : BOOL;
		VyrobaZacala : BOOL;
	END_STRUCT;
END_TYPE

(*//P2 - Šrobovanie//*)

TYPE
	P2_Srobovanie_typ : 	STRUCT
		CMD : P2_Srobovanie_CMD_typ;
		IN : P2_Srobovanie_IN_typ;
		OUT : P2_Srobovanie_OUT_typ;
		PAR : P2_Srobovanie_PAR_typ;
		STAV : P2_Srobovanie_STAV_typ;
		COM_IN : P2_Srobovanie_COM_IN_typ;
		COM_OUT : P2_Srobovanie_COM_OUT_typ;
		Automat : BOOL;
		Manual : BOOL;
		Reset : BOOL;
		KoniecCyklu : BOOL;
		ServoManipulOsX : ServoDriver;
		ServoManipulOsY : ServoDriver;
		ServoManipulOsZ_M4 : ServoDriver;
		Skrutkovacka_M4 : SkrutkovackaAtlasCopco_typ;
		Skrutkovacka_M5 : SkrutkovackaAtlasCopco_typ;
		Skrutkovacka_M6 : SkrutkovackaAtlasCopco_typ;
		SkrutSet_M4 : PickAndPlace;
		SkrutSet_M5 : ScrewLoading;
		SkrutSet_M6 : ScrewLoading;
	END_STRUCT;
	P2_Srobovanie_CMD_typ : 	STRUCT
		RR_Manipulator_OsX_VPRAVO : BOOL;
		RR_Manipulator_OsX_VLAVO : BOOL;
		RR_Manipulator_OsY_VPRED : BOOL;
		RR_Manipulator_OsY_VZAD : BOOL;
		RR_SkrutkovackaM4_OsZ_HORE : BOOL;
		RR_SkrutkovackaM4_OsZ_DOLE : BOOL;
		RR_PrisavanieSkrutkyM4_ON : BOOL;
		RR_PrisavanieSkrutkyM4_OFF : BOOL;
		RR_CistenieSkrutkovackyM6 : BOOL;
		RR_CistenieSkrutkovackyM5 : BOOL;
		RR_SkrutSetM6_Zasobnik_RUN : BOOL;
		RR_SkrutSetM6_PodajSkrutku : BOOL;
		RR_SkrutSetM6_VysunBrzdu : BOOL;
		RR_SkrutSetM5_Zasobnik_RUN : BOOL;
		RR_SkrutSetM5_PodajSkrutku : BOOL;
		RR_SkrutSetM5_VysunBrzdu : BOOL;
		RR_SkrutSetM4_Zasobnik_RUN : BOOL;
		RR_SkrutSetM4_Vibrolista_RUN : BOOL;
		RR_SkrutSetM4_PodajSkrutku : BOOL;
		RR_SkrutSetM4_OtocPodavac_Vstup : BOOL;
		RR_SkrutSetM4_OtocPodavac_Vystup : BOOL;
		RR_PolohujManipulator : BOOL;
		PodajSkrutku_M4 : BOOL;
		PodajSkrutku_M5 : BOOL;
		PodajSkrutku_M6 : BOOL;
	END_STRUCT;
	P2_Srobovanie_IN_typ : 	STRUCT
		ManipulOsX_LimSnimac_POS : BOOL; (*IS2_14*)
		ManipulOsX_LimSnimac_NEG : BOOL; (*IS2_13*)
		ManipulOsY_LimSnimac_POS : BOOL; (*IS2_16*)
		ManipulOsY_LimSnimac_NEG : BOOL; (*IS2_15*)
		ManipulOsZ_M4_LimSnimacHorny : BOOL; (*IS2_17*)
		ManipulOsZ_M4_LimSnimacSpodny : BOOL; (*IS2_18*)
		Skrutkovacka_M6_ZASUNUTA : BOOL; (*MS2_11*)
		Skrutkovacka_M5_ZASUNUTA : BOOL; (*MS2_10*)
		Skrutkovacka_M4_Vakum_OK : BOOL; (*S2_9*)
		NapajanieSkrutkovackyM6_OK : BOOL;
		NapajanieSkrutkovackyM4_OK : BOOL;
		NapajanieSkrutkovackyM5_OK : BOOL;
		NapajanieZasobnikaM6_OK : BOOL;
		NapajanieZasobnikaM5_OK : BOOL;
		NapajanieZasobnikaM4_OK : BOOL;
		NapajanieVibrolistyM4_OK : BOOL;
	END_STRUCT;
	P2_Srobovanie_OUT_typ : 	STRUCT
		Skrutkovacku_M6_VYSUN : BOOL; (*YV089_VT2*)
		Skrutkovacka_M6_Prisavanie_ON : BOOL; (*YV087_VT2*)
		Skrutkovacka_M6_Odvzdusn_ON : BOOL; (*YV088_VT2*)
		Skrutkovacku_M5_VYSUN : BOOL; (*YV096_VT2*)
		Skrutkovacka_M5_Prisavanie_ON : BOOL; (*YV094_VT2*)
		Skrutkovacka_M5_Odvzdusn_ON : BOOL; (*YV095_VT2*)
		Skrutkovacka_M4_Prisavanie_ON : BOOL; (*YV101_VT2*)
		Skrutkovacka_M4_Prisavanie_OFF : BOOL; (*YV102_VT2*)
		Skrutkovacka_M4_Odvzdusn_ON : BOOL; (*YV103_VT2*)
	END_STRUCT;
	P2_Srobovanie_PAR_typ : 	STRUCT
		ManipulOsZ_M4_AktualnaPozicia : REAL;
		Skrutkov_M5_AktualHodnVysunutia : UINT; (*IO-Link snímač*)
		Skrutkov_M5_RoundHodnotaREAL : REAL;
		Skrutkov_M6_AktualHodnVysunutia : UINT; (*IO-Link snímač*)
		Skrutkov_M6_RoundHodnotaREAL : REAL;
		ManipulOsX_AktualnaPozicia : REAL;
		ManipulOsY_AktualnaPozicia : REAL;
		RR_IndexPolohovaniaManipulatora : USINT;
		RR_TypModelu : STRING[2];
		ManipulOsX_JoggRychlost : REAL;
		ManipulOsY_JoggRychlost : REAL;
		ManipulOsZ_M4_JoggRychlost : REAL;
		M6_AtlasCopcoInputs : ARRAY[0..7]OF UDINT;
		M6_AtlasCopcoOutputs : ARRAY[0..7]OF UDINT;
		M5_AtlasCopcoInputs : ARRAY[0..7]OF UDINT;
		M5_AtlasCopcoOutputs : ARRAY[0..7]OF UDINT;
		M4_AtlasCopcoInputs : ARRAY[0..7]OF UDINT;
		M4_AtlasCopcoOutputs : ARRAY[0..7]OF UDINT;
	END_STRUCT;
	P2_Srobovanie_STAV_typ : 	STRUCT
		RR_Polohovanie_BUSY : BOOL;
		PoINIT : BOOL;
		Vysledok_Srobovania : STRING[2]; (*OK alebo NG*)
		M6_DosiahnutyMoment_REAL : REAL;
		M6_DosiahnutyMoment : UDINT;
		M6_Moment_ToleranciaMAX_REAL : REAL;
		M6_Moment_ToleranciaMAX : UDINT;
		M6_Moment_ToleranciaMIN_REAL : REAL;
		M6_Moment_ToleranciaMIN : UDINT;
		M6_DosiahnutyUhol : UINT;
		M6_Uhol_ToleranciaMAX_REAL : REAL;
		M6_Uhol_ToleranciaMAX : UDINT;
		M6_Uhol_ToleranciaMIN_REAL : REAL;
		M6_Uhol_ToleranciaMIN : UDINT;
		M5_DosiahnutyMoment_REAL : REAL;
		M5_DosiahnutyMoment : UDINT;
		M5_Moment_ToleranciaMAX_REAL : REAL;
		M5_Moment_ToleranciaMAX : UDINT;
		M5_Moment_ToleranciaMIN_REAL : REAL;
		M5_Moment_ToleranciaMIN : UDINT;
		M5_DosiahnutyUhol : UINT;
		M5_Uhol_ToleranciaMAX_REAL : REAL;
		M5_Uhol_ToleranciaMAX : UDINT;
		M5_Uhol_ToleranciaMIN_REAL : REAL;
		M5_Uhol_ToleranciaMIN : UDINT;
		M4_DosiahnutyMoment_REAL : REAL;
		M4_DosiahnutyMoment : UDINT;
		M4_Moment_ToleranciaMAX_REAL : REAL;
		M4_Moment_ToleranciaMAX : UDINT;
		M4_Moment_ToleranciaMIN_REAL : REAL;
		M4_Moment_ToleranciaMIN : UDINT;
		M4_DosiahnutyUhol : UINT;
		M4_Uhol_ToleranciaMAX_REAL : REAL;
		M4_Uhol_ToleranciaMAX : UDINT;
		M4_Uhol_ToleranciaMIN_REAL : REAL;
		M4_Uhol_ToleranciaMIN : UDINT;
		ManipulatorNadPodavacmi : BOOL;
		SkrutkaM6_READY : BOOL;
		SkrutkaM5_READY : BOOL;
		CistenieSkrutkovackyM5_BUSY : BOOL;
		CistenieSkrutkovackyM6_BUSY : BOOL;
	END_STRUCT;
	P2_Srobovanie_COM_IN_typ : 	STRUCT
		PresunManipulatora_VPRED : BOOL;
		PresunManipulatora_VZAD : BOOL;
		OdoberSkrutku_M4 : BOOL;
		Model45F_ZaskrutkujLavuM6 : BOOL;
		Model45F_ZaskrutkujPravuM6 : BOOL;
		Model45F_ZaskrutkujLavuM4 : BOOL;
		Model45F_ZaskrutkujPravuM4 : BOOL;
		Model5H_ZaskrutkujLavuM5 : BOOL;
		Model5H_ZaskrutkujPravuM5 : BOOL;
		Model5H_ZaskrutkujStrednuM4 : BOOL;
	END_STRUCT;
	P2_Srobovanie_COM_OUT_typ : 	STRUCT
		Stav_SkrutkovanieUkoncene : BOOL;
		Stav_PresunManipulUkonceny : BOOL;
		Stav_PoruchaSkrutkovania : BOOL;
	END_STRUCT;
END_TYPE

(*//P2 - Robot//*)

TYPE
	P2_Robot_typ : 	STRUCT
		CMD : P2_Robot_CMD_typ;
		IN : P2_Robot_IN_typ;
		OUT : P2_Robot_OUT_typ;
		PAR : P2_Robot_PAR_typ;
		STAV : P2_Robot_STAV_typ;
		COM_IN : P2_Robot_COM_IN_typ;
		COM_OUT : P2_Robot_COM_OUT_typ;
		Automat : BOOL;
		Manual : BOOL;
		Reset : BOOL;
		KoniecCyklu : BOOL;
	END_STRUCT;
	P2_Robot_CMD_typ : 	STRUCT
		New_Member : USINT;
	END_STRUCT;
	P2_Robot_IN_typ : 	STRUCT
		TypGripra_MvCase : BOOL; (*ROBHLA_013*)
		TypGripra_45F : BOOL; (*GRMECH_035*)
		TypGripra_5H : BOOL; (*GRMECH_036*)
		KodGripra_Bit0 : BOOL;
		KodGripra_Bit1 : BOOL;
		Model45F_Vakum_OK : BOOL; (*S2_6*)
		Model5H_Vakum_OK : BOOL; (*S2_7*)
		DokStanica_PritomGripraMvCase : BOOL; (*IS2_10 - Griper pre TopCover a MvCase*)
		DokStanica_PritomGripraBusbar45F : BOOL; (*IS2_11*)
		DokStanica_PritomGripraBusbar5H : BOOL; (*IS2_12*)
		GriperMvCase_Otvoreny : BOOL; (*IS2_37*)
		GriperMvCase_DrziPowerCP : BOOL; (*IS2_36*)
		GriperMvCase_DrziMvCase : BOOL; (*IS2_38*)
		GriperMvCase_Zatvoreny : BOOL;
		Griper45F_Otvoreny : BOOL;
		Griper45F_Zatvoreny : BOOL;
		Griper45F_DrziBusbary : BOOL;
		Griper5H_Otvoreny : BOOL;
		Griper5H_Zatvoreny : BOOL;
		Griper5H_DrziBusbary : BOOL;
	END_STRUCT;
	P2_Robot_OUT_typ : 	STRUCT
		OdistiGriper : BOOL; (*YV050_VT2*)
		ZaistiGriper : BOOL; (*YV049_VT2*)
		Griper_OTVOR : BOOL; (*YV051_VT2*)
		Griper_ZATVOR : BOOL; (*YV052_VT2*)
		Model45F_Vakum_ON : BOOL; (*YV054_VT2*)
		Model45F_Vakum_OFF : BOOL; (*YV055_VT2*)
		Model5H_Vakum_ON : BOOL; (*YV056_VT2*)
		Model5H_Vakum_OFF : BOOL; (*YV057_VT2*)
		PneuZamokUchopovaca_ODOMKNI : BOOL; (*YV053_VT2*)
	END_STRUCT;
	P2_Robot_PAR_typ : 	STRUCT
		Griper_Busbary45F_HodnOtvorenia : UINT; (*GRMECH_035 - IO-Link snímač*)
		Griper_Busbary5H_HodnOtvorenia : UINT; (*GRMECH_036 - IO-Link snímač*)
	END_STRUCT;
	P2_Robot_STAV_typ : 	STRUCT
		PoINIT : BOOL;
		DrziBusbar_4F : BOOL;
		DrziBusbar_5F : BOOL;
		DrziBusbar_5H : BOOL;
		Zvaranie_PrebiehaManipulacia : BOOL;
		Srobovanie_PrebiehaManipulacia : BOOL;
	END_STRUCT;
	P2_Robot_COM_IN_typ : 	STRUCT
		BYTE_IN : ARRAY[0..63]OF USINT; (*Z robota do PLC*)
		Stav_Busbary4F_Odobrate : BOOL;
		Stav_Busbary4F_Polozene : BOOL;
		Stav_Busbary5F_Odobrate : BOOL;
		Stav_Busbary5F_Polozene : BOOL;
		Stav_Busbary5H_Odobrate : BOOL;
		Stav_Busbary5H_Polozene : BOOL;
		Stav_PravyMvCase4F_Odobraty : BOOL;
		Stav_PravyMvCase4F_Polozeny : BOOL;
		Stav_LavyMvCase4F_Odobraty : BOOL;
		Stav_LavyMvCase4F_Polozeny : BOOL;
		Stav_PravyMvCase5F_Odobraty : BOOL;
		Stav_PravyMvCase5F_Polozeny : BOOL;
		Stav_LavyMvCase5F_Odobraty : BOOL;
		Stav_LavyMvCase5F_Polozeny : BOOL;
		Stav_PravyMvCase5H_Odobraty : BOOL;
		Stav_PravyMvCase5H_Polozeny : BOOL;
		Stav_LavyMvCase5H_Odobraty : BOOL;
		Stav_LavyMvCase5H_Polozeny : BOOL;
		Stav_TopCover4F_Odobraty : BOOL;
		Stav_TopCover4F_Polozeny : BOOL;
		Stav_TopCover5F_Odobraty : BOOL;
		Stav_TopCover5F_Polozeny : BOOL;
		Stav_TopCover5H_Odobraty : BOOL;
		Stav_TopCover5H_Polozeny : BOOL;
		Stav_Filter5H_Dotlaceny : BOOL;
		Stav_RobotOdparkovany : BOOL;
		Stav_RobotPoziciaCakania : BOOL;
		Stav_RobotBezpPozicia_Srobovanie : BOOL;
		Stav_RobotBezpPozicia_Zvaranie : BOOL;
		Stav_BusbaryUvolnene : BOOL;
		Stav_MotoryON : BOOL;
		Stav_MotoryOFF : BOOL;
		Stav_ProgramRUN : BOOL;
		Stav_RezimAUTOMAT : BOOL;
		Stav_RobotCS : BOOL;
		Stav_VystupyZresetovane : BOOL;
		Stav_Cistenie_PowerCP_Odobrate : BOOL;
		Stav_Cistenie_PowerCP_Polozene : BOOL;
		Stav_Cistenie_PowerCP_v_Cisteni : BOOL;
		Stav_Cistenie_Otacanie_Ukoncene : BOOL;
		Stav_Griper4F5F_Vymeneny : BOOL;
		Stav_Griper5H_Vymeneny : BOOL;
		Stav_GriperCistenia_Vymeneny : BOOL;
		Stav_RobotOdoberaCover : BOOL;
	END_STRUCT;
	P2_Robot_COM_OUT_typ : 	STRUCT
		BYTE_OUT : ARRAY[0..63]OF USINT; (*Z PLC do Robota*)
		ManipSrobovania_BezpecnaPozicia : BOOL;
		Zvaranie_BezpecnaPozicia : BOOL;
		Cistenie_BezpecnaPozicia : BOOL;
		Odober_Busbary4F : BOOL;
		Poloz_Busbary4F : BOOL;
		Odober_Busbary5F : BOOL;
		Poloz_Busbary5F : BOOL;
		Odober_Busbary5H : BOOL;
		Poloz_Busbary5H : BOOL;
		Odober_PravyMvCase4F : BOOL;
		Poloz_PravyMvCase4F : BOOL;
		Odober_LavyMvCase4F : BOOL;
		Poloz_LavyMvCase4F : BOOL;
		Odober_PravyMvCase5F : BOOL;
		Poloz_PravyMvCase5F : BOOL;
		Odober_LavyMvCase5F : BOOL;
		Poloz_LavyMvCase5F : BOOL;
		Odober_PravyMvCase5H : BOOL;
		Poloz_PravyMvCase5H : BOOL;
		Odober_LavyMvCase5H : BOOL;
		Poloz_LavyMvCase5H : BOOL;
		Odober_TopCover4F : BOOL;
		Poloz_TopCover4F : BOOL;
		Odober_TopCover5F : BOOL;
		Poloz_TopCover5F : BOOL;
		Odober_TopCover5H : BOOL;
		Poloz_TopCover5H : BOOL;
		Dotlac_Filter5H : BOOL;
		Cistenie_OdoberPowerCP_4F : BOOL;
		Cistenie_OdoberPowerCP_5F : BOOL;
		Cistenie_OdoberPowerCP_5H : BOOL;
		Cistenie_OtacajPowerCP : BOOL;
		Cistenie_PolozPowerCP_4F : BOOL;
		Cistenie_PolozPowerCP_5F : BOOL;
		Cistenie_PolozPowerCP_5H : BOOL;
		Presun_CakaciaPozicia : BOOL;
		UvolniBusbary : BOOL;
		Odparkovanie : BOOL;
		ZapniMotory : BOOL;
		VypniMotory : BOOL;
		PP_na_Main : BOOL;
		Reset_CS : BOOL;
		StartProgramu : BOOL;
		StartProgramuMain : BOOL;
		StopProgramu : BOOL;
		Griper4F_Otvoreny : BOOL;
		Griper4F_Zatvoreny : BOOL;
		Griper4F_DrziBusbary : BOOL;
		Griper5H_Otvoreny : BOOL;
		Griper5H_Zatvoreny : BOOL;
		Griper5H_DrziBusbary : BOOL;
		GriperMvCase_Zatvoreny : BOOL; (*Griper pre MV Case a Top Cover*)
		GriperMvCase_Otvoreny : BOOL; (*Griper pre MV Case a Top Cover*)
		GriperMvCase_DrziPowerCP : BOOL;
		GriperMvCase_DrziMVcase : BOOL;
		ZmenaGripra_4F5F : BOOL;
		ZmenaGripra_5H : BOOL;
		ZmenaGripra_Cistenie : BOOL;
		ZopakujOdoberanie : BOOL;
	END_STRUCT;
END_TYPE

(*//P2 - Stoper zvarania//*)

TYPE
	P2_StoperZvarania_typ : 	STRUCT
		CMD : P2_StoperZvarania_CMD_typ;
		IN : P2_StoperZvarania_IN_typ;
		OUT : P2_StoperZvarania_OUT_typ;
		PAR : P2_StoperZvarania_PAR_typ;
		STAV : P2_StoperZvarania_STAV_typ;
		RFID_hlava : SickHeads;
		Automat : BOOL;
		Manual : BOOL;
		Reset : BOOL;
		KoniecCyklu : BOOL;
	END_STRUCT;
	P2_StoperZvarania_CMD_typ : 	STRUCT
		RR_VysunCentrovanie : BOOL;
	END_STRUCT;
	P2_StoperZvarania_IN_typ : 	STRUCT
		Centrovanie_VYSUNUTE : BOOL; (*IS2_6*)
		Centrovanie_ZASUNUTE : BOOL; (*IS2_7*)
	END_STRUCT;
	P2_StoperZvarania_OUT_typ : 	STRUCT
		ZasunStoper : BOOL; (*YV045_VT2*)
		Centrovanie_VYSUN : BOOL; (*YV046_VT2*)
		Centrovanie_ZASUN : BOOL; (*YV047_VT2*)
	END_STRUCT;
	P2_StoperZvarania_PAR_typ : 	STRUCT
		CisloPaletky_STRING : STRING[2];
		IndexFotky : USINT;
		CisloPaletky : USINT;
	END_STRUCT;
	P2_StoperZvarania_STAV_typ : 	STRUCT
		PoINIT : BOOL;
		PrebiehaVyvezeniePaletky : BOOL;
		VstupnaKamerovaKontrola : BOOL;
		VyrobaZacala : BOOL;
	END_STRUCT;
END_TYPE

(*//P2 - Zvaranie//*)

TYPE
	P2_Zvaranie_typ : 	STRUCT
		CMD : P2_Zvaranie_CMD_typ;
		IN : P2_Zvaranie_IN_typ;
		OUT : P2_Zvaranie_OUT_typ;
		PAR : P2_Zvaranie_PAR_typ;
		STAV : P2_Zvaranie_STAV_typ;
		COM_IN : P2_Zvaranie_COM_IN_typ;
		COM_OUT : P2_Zvaranie_COM_OUT_typ;
		Automat : BOOL;
		Manual : BOOL;
		Reset : BOOL;
		KoniecCyklu : BOOL;
		ServoZdvihuZvarania : ServoDriver;
	END_STRUCT;
	P2_Zvaranie_CMD_typ : 	STRUCT
		RR_ZdvihZvarania_HORE : BOOL;
		RR_ZdvihZvarania_DOLE : BOOL;
		RR_SekvenciaZvarania_START : BOOL;
		RR_Presun_VPRAVO : BOOL;
		RR_Presun_VLAVO : BOOL;
	END_STRUCT;
	P2_Zvaranie_IN_typ : 	STRUCT
		ZdvihZvarania_HornyLimSnimac : BOOL; (*IS2_19*)
		ZvaraniePresunute_VPRAVO : BOOL; (*IS2_20*)
		ZvaraniePresunute_VLAVO : BOOL; (*IS2_21*)
		NapajanieZvaracky_OK : BOOL;
		ZvarackaStav_RUN : BOOL;
		ZvarackaStav_READY : BOOL;
	END_STRUCT;
	P2_Zvaranie_OUT_typ : 	STRUCT
		PresunZvaranie_VPRAVO : BOOL; (*YV063_VT2*)
		PresunZvarania_VLAVO : BOOL; (*YV064_VT2*)
		Zvaracka_START : BOOL;
		Zvaracka_RESET : BOOL;
	END_STRUCT;
	P2_Zvaranie_PAR_typ : 	STRUCT
		ZdvihZvarania_JoggRychlost : REAL;
	END_STRUCT;
	P2_Zvaranie_STAV_typ : 	STRUCT
		PoINIT : BOOL;
		Vysledok_Zvarania : STRING[2]; (*OK alebo NG*)
		RR_SekvenciaZvarania_BUSY : BOOL;
	END_STRUCT;
	P2_Zvaranie_COM_IN_typ : 	STRUCT
		Zvaranie_START : BOOL;
		Zatlacanie_START : BOOL;
	END_STRUCT;
	P2_Zvaranie_COM_OUT_typ : 	STRUCT
		Stav_ZvaranieUkoncene : BOOL;
		Stav_ZatlacenieUkoncene : BOOL;
	END_STRUCT;
END_TYPE

(*//P2 - Čistenie//*)

TYPE
	P2_Cistenie_typ : 	STRUCT
		CMD : P2_Cistenie_CMD_typ;
		IN : P2_Cistenie_IN_typ;
		OUT : P2_Cistenie_OUT_typ;
		PAR : P2_Cistenie_PAR_typ;
		STAV : P2_Cistenie_STAV_typ;
		COM_IN : P2_Cistenie_COM_IN_typ;
		COM_OUT : P2_Cistenie_COM_OUT_typ;
		Automat : BOOL;
		Manual : BOOL;
		Reset : BOOL;
		KoniecCyklu : BOOL;
	END_STRUCT;
	P2_Cistenie_CMD_typ : 	STRUCT
		RR_Cistenie_OTVOR : BOOL;
		RR_Cistenie_ZATVOR : BOOL;
	END_STRUCT;
	P2_Cistenie_IN_typ : 	STRUCT
		Dvere_OTVORENE : BOOL; (*MS2_1*)
		Dvere_ZATVORENE : BOOL; (*MS2_2*)
		Vakum_OK : BOOL; (*S2_8*)
		Ionizator_Alarm1 : BOOL;
		Ionizator_Alarm2 : BOOL;
		Ionizator_Alarm3 : BOOL;
	END_STRUCT;
	P2_Cistenie_OUT_typ : 	STRUCT
		Ionizator_OFF : BOOL; (*YV060_VT2*)
		VzduchPreIonizator_ON : BOOL;
		Dvere_ZATVOR : BOOL;
		Dvere_OTVOR : BOOL;
		Odsavanie_ON : BOOL; (*YV061_VT2*)
		OdsavanieOfuk_ON : BOOL; (*YV062_VT2*)
	END_STRUCT;
	P2_Cistenie_PAR_typ : 	STRUCT
		PAR_0 : USINT;
	END_STRUCT;
	P2_Cistenie_STAV_typ : 	STRUCT
		PoINIT : BOOL;
	END_STRUCT;
	P2_Cistenie_COM_IN_typ : 	STRUCT
		Cistenie_START : BOOL;
	END_STRUCT;
	P2_Cistenie_COM_OUT_typ : 	STRUCT
		Stav_CistenieUkoncene : BOOL;
	END_STRUCT;
END_TYPE

(***********************************Pracovisko 3****************************************************************)

TYPE
	P3_Pracovisko_typ : 	STRUCT
		IN : P3_Pracovisko_IN_typ;
		OUT : P3_Pracovisko_OUT_typ;
		PAR : P3_Pracovisko_PAR_typ;
		STAV : P3_Pracovisko_STAV_typ;
		COM_Weidmuller : P3_COM_Weidmuller_typ;
		COM_Festo : P3_COM_Festo_typ;
		COM_VentilovyTerminal : ARRAY[0..9]OF USINT;
		Automat : BOOL;
		Manual : BOOL;
		Reset : BOOL;
		KoniecCyklu : BOOL;
	END_STRUCT;
	P3_Pracovisko_IN_typ : 	STRUCT
		TlakVzduchu_OK : BOOL; (*S3_7*)
		ModulWeidmuller_IO_KomOK : BOOL;
		VentilovyTerminal_KomOK : BOOL;
		Skrutkovacka_K40_KomOK : BOOL;
		Skrutkovacka_M5_KomOK : BOOL;
		ModulFesto_IO_KomOK : BOOL;
		ServoManipulatorOsY_KomOK : BOOL;
		ServoManipulatorOsZ_M5_KomOK : BOOL;
		Kamery_ControlUnit_KomOK : BOOL;
		LeakageTesterA_KomOK : BOOL;
		LeakageTesterB_KomOK : BOOL;
		StavPrepatovejOchrany_OK : BOOL;
		PredneDvereLave_PritomnAdaptera : BOOL; (*EZ 3.1*)
		PredneDverePrave_PritomnAdaptera : BOOL; (*EZ 3.2*)
		ZadneDvereLave_PritomnAdaptera : BOOL; (*EZ 3.3*)
		ZadneDverePrave_PritomnAdaptera : BOOL; (*EZ 3.4*)
	END_STRUCT;
	P3_Pracovisko_OUT_typ : 	STRUCT
		Majak_ZeleneSvetlo_ON : BOOL;
		Majak_OranzoveSvetlo_ON : BOOL;
		Majak_CerveneSvetlo_ON : BOOL;
		Majak_Hukacka_ON : BOOL;
		OsvetlenieBunky_ON : BOOL;
		Osvetlenie_CAM13_ON : BOOL;
		ZdvizkyPneuZamok_ODOMKNI : BOOL; (*YV166_VT3*)
		PredneDvereLave_ZAMKNI : BOOL; (*EZ 3.1*)
		PredneDverePrave_ZAMKNI : BOOL; (*EZ 3.2*)
		ZadneDvereLave_ZAMKNI : BOOL; (*EZ 3.3*)
		ZadneDverePrave_ZAMKNI : BOOL; (*EZ 3.4*)
		Ventilator_ON : BOOL;
	END_STRUCT;
	P3_Pracovisko_PAR_typ : 	STRUCT
		New_Member : USINT;
	END_STRUCT;
	P3_Pracovisko_STAV_typ : 	STRUCT
		Automat : BOOL;
		Manual : BOOL;
		PoINIT : BOOL;
		READY : BOOL;
		PORUCHA : BOOL;
		HardwareBunky_OK : BOOL;
		Porucha_ST1 : BOOL; (*Šrobovanie*)
		Porucha_ST2 : BOOL; (*HV test*)
		Porucha_ST3 : BOOL; (*Zdvizka pred Leakage testom A*)
		Porucha_ST4 : BOOL; (*Zdvizka pred Leakage testom B*)
		Porucha_ST5 : BOOL; (*Leakage test A*)
		Porucha_ST6 : BOOL; (*Leakage test B*)
		Porucha_ST7 : BOOL; (*Zdvizka za Leakage testom A*)
		Porucha_ST8 : BOOL; (*Zdvizka za Leakage testom B*)
		SkrutkovackyZasunute : BOOL;
		UkoncenieCyklu_BUSY : BOOL;
		HVtest_Zasunuty : BOOL;
		LeakageTestA_Zasunuty : BOOL;
		LeakageTestB_Zasunuty : BOOL;
		PredneDvereZamknute : BOOL;
		ZadneDvereZamknute : BOOL;
	END_STRUCT;
	P3_COM_Weidmuller_typ : 	STRUCT
		AB3_5_8DI : USINT;
		AB3_6_8DI : USINT;
		AB3_7_8DI : USINT;
		AB3_8_8DI : USINT;
		AB3_9_8DO : USINT;
		AB3_10_8DO : USINT;
		AB3_12_8DO : USINT;
	END_STRUCT;
	P3_COM_Festo_typ : 	STRUCT
		DM3_1_4DI : ARRAY[0..3]OF BOOL;
		DM3_1_4DO : ARRAY[0..3]OF BOOL;
		DI3_1_8DI : ARRAY[0..7]OF BOOL;
		DI3_2_8DI : ARRAY[0..7]OF BOOL;
		DI3_3_8DI : ARRAY[0..7]OF BOOL;
		DI3_4_8DI : ARRAY[0..7]OF BOOL;
		DI3_5_8DI : ARRAY[0..7]OF BOOL;
		DI3_6_8DI : ARRAY[0..7]OF BOOL;
		DI3_7_8DI : ARRAY[0..7]OF BOOL;
		DI3_8_8DI : ARRAY[0..7]OF BOOL;
		DI3_9_8DI : ARRAY[0..7]OF BOOL;
		DI3_10_8DI : ARRAY[0..7]OF BOOL;
		DS3_1_Port0_IN : ARRAY[0..31]OF USINT;
		DS3_1_Port0_OUT : ARRAY[0..31]OF USINT;
		DS3_1_Port1_IN : ARRAY[0..31]OF USINT;
		DS3_1_Port1_OUT : ARRAY[0..31]OF USINT;
		DS3_1_Port2_IN : ARRAY[0..31]OF USINT;
		DS3_1_Port2_OUT : ARRAY[0..31]OF USINT;
		DS3_1_Port3_IN : ARRAY[0..31]OF USINT;
		DS3_1_Port3_OUT : ARRAY[0..31]OF USINT;
		DS3_2_Port0_IN : ARRAY[0..1]OF USINT;
		DS3_2_Port0_OUT : ARRAY[0..1]OF USINT;
		DS3_2_Port1_IN : ARRAY[0..1]OF USINT;
		DS3_2_Port1_OUT : ARRAY[0..1]OF USINT;
		DS3_2_Port2_IN : ARRAY[0..1]OF USINT;
		DS3_2_Port2_OUT : ARRAY[0..1]OF USINT;
	END_STRUCT;
END_TYPE

(*//P3 - Dopravníky//*)

TYPE
	P3_Dopravniky_typ : 	STRUCT
		IN : P3_Dopravniky_IN_typ;
		OUT : P3_Dopravniky_OUT_typ;
		PAR : P3_Dopravniky_PAR_typ;
		STAV : P3_Dopravniky_STAV_typ;
		Automat : BOOL;
		Manual : BOOL;
		Reset : BOOL;
		KoniecCyklu : BOOL;
	END_STRUCT;
	P3_Dopravniky_IN_typ : 	STRUCT
		StavRiadeniaVratnehoDoprav_READY : BOOL; (*M3_12*)
		StavRiadPredDopravBunky_READY : BOOL; (*M3_8*)
		StavRiadZadnDopravBunky_READY : BOOL; (*M3_11*)
		StavRiadeniaPriecnDoprav1_READY : BOOL; (*M3_9*)
		StavRiadeniaPriecnDoprav2_READY : BOOL; (*M3_10*)
		TeplotaMotoraVratnehoDoprav_OK : BOOL; (*M3_12*)
		TeplotaMotoraPredDopravBunky_OK : BOOL; (*M3_8*)
		TeplotaMotoraZadnDopravBunky_OK : BOOL; (*M3_11*)
		TeplotaMotoraPriecnDoprav1_OK : BOOL; (*M3_9*)
		TeplotaMotoraPriecnDoprav2_OK : BOOL; (*M3_10*)
	END_STRUCT;
	P3_Dopravniky_OUT_typ : 	STRUCT
		PrednyDopravnikBunky_ON : BOOL; (*M3_8*)
		ZadnyDopravnikBunky_ON : BOOL; (*M3_11*)
		VratnyDopravnik_ON : BOOL; (*M3_12*)
		PriecnyDopravnik1_VPRED : BOOL; (*M3_9 - Smerom na trať B*)
		PriecnyDopravnik2_VPRED : BOOL; (*M3_10 - Smerom na trať B*)
		PriecnyDopravnik2_VZAD : BOOL; (*M3_10 - Smerom na trať A*)
	END_STRUCT;
	P3_Dopravniky_PAR_typ : 	STRUCT
		New_Member : USINT;
	END_STRUCT;
	P3_Dopravniky_STAV_typ : 	STRUCT
		PoINIT : BOOL;
	END_STRUCT;
END_TYPE

(*//P3 - Spodný stoper//*)

TYPE
	P3_SpodnyStoper_typ : 	STRUCT
		IN : P3_SpodnyStoper_IN_typ;
		OUT : P3_SpodnyStoper_OUT_typ;
		PAR : P3_SpodnyStoper_PAR_typ;
		STAV : P3_SpodnyStoper_STAV_typ;
		Automat : BOOL;
		Manual : BOOL;
		Reset : BOOL;
		KoniecCyklu : BOOL;
	END_STRUCT;
	P3_SpodnyStoper_IN_typ : 	STRUCT
		PritomnostPaletky : BOOL; (*IS3_26*)
		ZaplnenieDopravnika : BOOL; (*IS3_27*)
	END_STRUCT;
	P3_SpodnyStoper_OUT_typ : 	STRUCT
		ZasunStoper : BOOL; (*YV125_VT3*)
	END_STRUCT;
	P3_SpodnyStoper_PAR_typ : 	STRUCT
		New_Member : USINT;
	END_STRUCT;
	P3_SpodnyStoper_STAV_typ : 	STRUCT
		PoINIT : BOOL;
		PrebiehaVyvezeniePaletky : BOOL;
	END_STRUCT;
END_TYPE

(*//P3 - Stoper šrobovania//*)

TYPE
	P3_StoperSrobovania_typ : 	STRUCT
		CMD : P3_StoperSrobovania_CMD_typ;
		IN : P3_StoperSrobovania_IN_typ;
		OUT : P3_StoperSrobovania_OUT_typ;
		PAR : P3_StoperSrobovania_PAR_typ;
		STAV : P3_StoperSrobovania_STAV_typ;
		RFID_hlava : SickHeads;
		Automat : BOOL;
		Manual : BOOL;
		Reset : BOOL;
		KoniecCyklu : BOOL;
	END_STRUCT;
	P3_StoperSrobovania_CMD_typ : 	STRUCT
		RR_VysunCentrovanie : BOOL;
	END_STRUCT;
	P3_StoperSrobovania_IN_typ : 	STRUCT
		Centrovanie_VYSUNUTE : BOOL; (*IS3_5*)
		Centrovanie_ZASUNUTE : BOOL; (*IS3_6*)
	END_STRUCT;
	P3_StoperSrobovania_OUT_typ : 	STRUCT
		ZasunStoper : BOOL; (*YV104_VT3*)
		Centrovanie_VYSUN : BOOL; (*YV105_VT3*)
		Centrovanie_ZASUN : BOOL; (*YV106_VT3*)
	END_STRUCT;
	P3_StoperSrobovania_PAR_typ : 	STRUCT
		CisloPaletky_STRING : STRING[2];
		IndexFotky : USINT;
		CisloPaletky : USINT;
	END_STRUCT;
	P3_StoperSrobovania_STAV_typ : 	STRUCT
		PoINIT : BOOL;
		PrebiehaVyvezeniePaletky : BOOL;
		VstupnaKamerovaKontrola : BOOL;
		VyrobaZacala : BOOL;
	END_STRUCT;
END_TYPE

(*//P3 - Šrobovanie//*)

TYPE
	P3_Srobovanie_typ : 	STRUCT
		CMD : P3_Srobovanie_CMD_typ;
		IN : P3_Srobovanie_IN_typ;
		OUT : P3_Srobovanie_OUT_typ;
		PAR : P3_Srobovanie_PAR_typ;
		STAV : P3_Srobovanie_STAV_typ;
		COM_IN : P3_Srobovanie_COM_IN_typ;
		COM_OUT : P3_Srobovanie_COM_OUT_typ;
		Automat : BOOL;
		Manual : BOOL;
		Reset : BOOL;
		KoniecCyklu : BOOL;
		ServoManipulOsY : ServoDriver;
		ServoManipulOsZ_M5 : ServoDriver;
		Skrutkovacka_K40 : SkrutkovackaAtlasCopco_typ;
		Skrutkovacka_M5 : SkrutkovackaAtlasCopco_typ;
		SkrutSet_K40 : ScrewLoading;
		SkrutSet_M5 : PickAndPlace;
	END_STRUCT;
	P3_Srobovanie_CMD_typ : 	STRUCT
		RR_Manipulator_OsY_VPRED : BOOL;
		RR_Manipulator_OsY_VZAD : BOOL;
		RR_M45F_PresunNaPozSkrutkov : BOOL;
		RR_M5H_PresunNaPozSkrutkov : BOOL;
		RR_PrisavanieSkrutkyM5_ON : BOOL;
		RR_PrisavanieSkrutkyM5_OFF : BOOL;
		RR_SkrutkovackaM5_OsZ_HORE : BOOL;
		RR_SkrutkovackaM5_OsZ_DOLE : BOOL;
		RR_CistenieSkrutkovackyK40 : BOOL;
		RR_SkrutSetK40_Zasobnik_RUN : BOOL;
		RR_SkrutSetK40_PodajSkrutku : BOOL;
		RR_SkrutSetK40_VysunBrzdu : BOOL;
		RR_SkrutSetM5_Zasobnik_RUN : BOOL;
		RR_SkrutSetM5_Vibrolista_RUN : BOOL;
		RR_SkrutSetM5_PodajSkrutku : BOOL;
		RR_SkrutSetM5_OtocPodavac_Vstup : BOOL;
		RR_SkrutSetM5_OtocPodavac_Vystup : BOOL;
		RR_PolohujManipulator : BOOL;
		PodajSkrutku_K40 : BOOL;
		PodajSkrutku_M5 : BOOL;
	END_STRUCT;
	P3_Srobovanie_IN_typ : 	STRUCT
		ManipulOsY_LimSnimac_POS : BOOL; (*IS3_2*)
		ManipulOsY_LimSnimac_NEG : BOOL; (*IS3_1*)
		ManipulOsZ_M5_LimSnimacHorny : BOOL; (*IS3_3*)
		ManipulOsZ_M5_LimSnimacSpodny : BOOL; (*IS3_4*)
		Skrutkovacka_K40_ZASUNUTA : BOOL; (*MS3_6*)
		Skrutkovacka_M5_Vakum_OK : BOOL; (*S3_6*)
		NapajanieSkrutkovackyK40_OK : BOOL;
		NapajanieSkrutkovackyM5_OK : BOOL;
		NapajanieZasobnikaK40_OK : BOOL;
		NapajanieZasobnikaM5_OK : BOOL;
		NapajanieVibrolistyM5_OK : BOOL;
	END_STRUCT;
	P3_Srobovanie_OUT_typ : 	STRUCT
		Skrutkovacku_K40_VYSUN : BOOL; (*YV158_VT3*)
		Skrutkovacka_K40_Prisavanie_ON : BOOL; (*YV156_VT3*)
		Skrutkovacka_K40_Odvzdusn_ON : BOOL; (*YV157_VT3*)
		Skrutkovacka_M5_Prisavanie_ON : BOOL; (*YV163_VT3*)
		Skrutkovacka_M5_Prisavanie_OFF : BOOL; (*YV164_VT3*)
		Skrutkovacka_M5_Odvzdusn_ON : BOOL; (*YV165_VT3*)
	END_STRUCT;
	P3_Srobovanie_PAR_typ : 	STRUCT
		Skrutkov_K40_AktualHodnVysunutia : UINT; (*IO-Link snímač*)
		Skrutkov_K40_RoundHodnotaREAL : REAL;
		ManipulOsY_AktualnaPozicia : REAL;
		ManipulOsZ_M5_AktualnaPozicia : REAL;
		RR_IndexPolohovaniaManipulatora : USINT;
		ManipulOsY_JoggRychlost : REAL;
		ManipulOsZ_M5_JoggRychlost : REAL;
		K40_AtlasCopcoInputs : ARRAY[0..7]OF UDINT;
		K40_AtlasCopcoOutputs : ARRAY[0..7]OF UDINT;
		M5_AtlasCopcoInputs : ARRAY[0..7]OF UDINT;
		M5_AtlasCopcoOutputs : ARRAY[0..7]OF UDINT;
	END_STRUCT;
	P3_Srobovanie_STAV_typ : 	STRUCT
		PoINIT : BOOL;
		Vysledok_SrobovaniaK40 : STRING[2]; (*OK alebo NG*)
		Vysledok_SrobovaniaM5 : STRING[2]; (*OK alebo NG*)
		RR_Polohovanie_BUSY : BOOL;
		K40_DosiahnutyMoment_REAL : REAL;
		K40_DosiahnutyMoment : UDINT;
		K40_Moment_ToleranciaMAX_REAL : REAL;
		K40_Moment_ToleranciaMAX : UDINT;
		K40_Moment_ToleranciaMIN_REAL : REAL;
		K40_Moment_ToleranciaMIN : UDINT;
		K40_DosiahnutyUhol : UINT;
		K40_Uhol_ToleranciaMAX_REAL : REAL;
		K40_Uhol_ToleranciaMAX : UDINT;
		K40_Uhol_ToleranciaMIN_REAL : REAL;
		K40_Uhol_ToleranciaMIN : UDINT;
		M5_DosiahnutyMoment_REAL : REAL;
		M5_DosiahnutyMoment : UDINT;
		M5_Moment_ToleranciaMAX_REAL : REAL;
		M5_Moment_ToleranciaMAX : UDINT;
		M5_Moment_ToleranciaMIN_REAL : REAL;
		M5_Moment_ToleranciaMIN : UDINT;
		M5_DosiahnutyUhol : UINT;
		M5_Uhol_ToleranciaMAX_REAL : REAL;
		M5_Uhol_ToleranciaMAX : UDINT;
		M5_Uhol_ToleranciaMIN_REAL : REAL;
		M5_Uhol_ToleranciaMIN : UDINT;
		SkrutkaK40_READY : BOOL;
		CistenieSkrutkovackyK40_BUSY : BOOL;
	END_STRUCT;
	P3_Srobovanie_COM_IN_typ : 	STRUCT
		PresunManipulatora_VPRED : BOOL;
		PresunManipulatora_VZAD : BOOL;
		Model45F_ZaskrutkujSkrutky : BOOL;
		Model5H_ZaskrutkujSkrutky : BOOL;
	END_STRUCT;
	P3_Srobovanie_COM_OUT_typ : 	STRUCT
		Stav_SkrutkovanieUkoncene : BOOL;
		Stav_PresunManipulUkonceny : BOOL;
		Stav_PoruchaSkrutkovania : BOOL;
	END_STRUCT;
END_TYPE

(*//P3 - HV test//*)

TYPE
	P3_HV_Test_typ : 	STRUCT
		CMD : P3_HV_Test_CMD_typ;
		IN : P3_HV_Test_IN_typ;
		OUT : P3_HV_Test_OUT_typ;
		PAR : P3_HV_Test_PAR_typ;
		STAV : P3_HV_Test_STAV_typ;
		RFID_hlava : SickHeads;
		Automat : BOOL;
		Manual : BOOL;
		Reset : BOOL;
		KoniecCyklu : BOOL;
	END_STRUCT;
	P3_HV_Test_CMD_typ : 	STRUCT
		RR_ZatvorTester : BOOL;
		StartTestovania : BOOL;
		RR_VysunCentrovanie : BOOL;
		RR_VysunPruzenieKontaktov : BOOL;
		OpatovnyTest : BOOL;
	END_STRUCT;
	P3_HV_Test_IN_typ : 	STRUCT
		Centrovanie_VYSUNUTE : BOOL; (*MS3_12*)
		Centrovanie_ZASUNUTE : BOOL; (*MS3_11*)
		SpodneKontakty_ZASUNUTE : BOOL; (*MS3_13*)
		SpodneKontakty_VYSUNUTE : BOOL; (*MS3_14*)
		HorneKontakty_ZASUNUTE : BOOL; (*MS3_10*)
		HorneKontakty_VYSUNUTE : BOOL; (*MS3_9*)
		TypKonektoru_4F : BOOL;
		TypKonektoru_5F_5H : BOOL;
	END_STRUCT;
	P3_HV_Test_OUT_typ : 	STRUCT
		ZasunStoper : BOOL; (*YV107_VT3*)
		Centrovanie_VYSUN : BOOL; (*YV138_VT3*)
		Centrovanie_ZASUN : BOOL; (*YV139_VT3*)
		SpodneKontakty_ZASUN : BOOL; (*YV140_VT3*)
		SpodneKontakty_VYSUN : BOOL; (*YV141_VT3*)
		HorneKontakty_ZASUN : BOOL; (*YV135_VT3*)
		HorneKontakty_VYSUN : BOOL; (*YV134_VT3*)
		PritlacenieKontaktovTestera_ON : BOOL; (*YV142_VT3*)
		PruzenieHornychKontaktov_VYSUN : BOOL;
		PruzenieHornychKontaktov_ZASUN : BOOL;
	END_STRUCT;
	P3_HV_Test_PAR_typ : 	STRUCT
		CisloPaletky_STRING : STRING[2];
		CisloPortuKlienta : UINT;
	END_STRUCT;
	P3_HV_Test_STAV_typ : 	STRUCT
		PoINIT : BOOL;
		PrebiehaVyvezeniePaletky : BOOL;
		TestovanieUkoncene : BOOL;
		TesterNeodpoveda : BOOL;
		Vysledok_HV_Testu : STRING[2]; (*OK alebo NG*)
		NameranyCas_InitTestera : TIME;
		NameranyCas_PoslanieQRkodu : TIME;
		NameranyCas_CelkovyCasTestovania : TIME;
		RR_SekvenciaTestera_BUSY : BOOL;
		PaletkaOznacena_NG : BOOL;
	END_STRUCT;
END_TYPE

(*//P3 - Zdvižka pred Leakage Testom A//*)

TYPE
	P3_ZdvizkaPredLeakTestA_typ : 	STRUCT
		IN : P3_ZdvizkaPredLeakTestA_IN_typ;
		OUT : P3_ZdvizkaPredLeakTestA_OUT_typ;
		PAR : P3_ZdvizkaPredLeakTestA_PAR_typ;
		STAV : P3_ZdvizkaPredLeakTestA_STAV_typ;
		Automat : BOOL;
		Manual : BOOL;
		Reset : BOOL;
		KoniecCyklu : BOOL;
	END_STRUCT;
	P3_ZdvizkaPredLeakTestA_IN_typ : 	STRUCT
		PritomnostPaletky : BOOL; (*IS3_10*)
		Zdvizka_HornaPoloha : BOOL; (*IS3_8*)
		Zdvizka_SpodnaPoloha : BOOL; (*IS3_7*)
		Zdvizka_StrednaPoloha : BOOL; (*IS3_9*)
	END_STRUCT;
	P3_ZdvizkaPredLeakTestA_OUT_typ : 	STRUCT
		Zdvizku_ZASUN : BOOL; (*YV108_VT3*)
		Zdvizku_VYSUN : BOOL; (*YV109_VT3*)
		TlmicPaletky_VYSUN : BOOL; (*YV110_VT3*)
	END_STRUCT;
	P3_ZdvizkaPredLeakTestA_PAR_typ : 	STRUCT
		New_Member : USINT;
	END_STRUCT;
	P3_ZdvizkaPredLeakTestA_STAV_typ : 	STRUCT
		PoINIT : BOOL;
		PrebiehaVyvezeniePaletkyNaTratA : BOOL;
		PrebiehaVyvezeniePaletkyNaTratB : BOOL;
	END_STRUCT;
END_TYPE

(*//P3 - Zdvižka pred Leakage Testom B//*)

TYPE
	P3_ZdvizkaPredLeakTestB_typ : 	STRUCT
		IN : P3_ZdvizkaPredLeakTestB_IN_typ;
		OUT : P3_ZdvizkaPredLeakTestB_OUT_typ;
		PAR : P3_ZdvizkaPredLeakTestB_PAR_typ;
		STAV : P3_ZdvizkaPredLeakTestB_STAV_typ;
		Automat : BOOL;
		Manual : BOOL;
		Reset : BOOL;
		KoniecCyklu : BOOL;
	END_STRUCT;
	P3_ZdvizkaPredLeakTestB_IN_typ : 	STRUCT
		PritomnostPaletky : BOOL; (*IS3_15*)
		PoziciaPaletky_OK : BOOL; (*IS3_14*)
		Zdvizka_HornaPoloha : BOOL; (*IS3_12*)
		Zdvizka_SpodnaPoloha : BOOL; (*IS3_11*)
		Zdvizka_StrednaPoloha : BOOL; (*IS3_13*)
	END_STRUCT;
	P3_ZdvizkaPredLeakTestB_OUT_typ : 	STRUCT
		Zdvizku_ZASUN : BOOL; (*YV111_VT3*)
		Zdvizku_VYSUN : BOOL; (*YV112_VT3*)
	END_STRUCT;
	P3_ZdvizkaPredLeakTestB_PAR_typ : 	STRUCT
		New_Member : USINT;
	END_STRUCT;
	P3_ZdvizkaPredLeakTestB_STAV_typ : 	STRUCT
		PoINIT : BOOL;
		PrebiehaVyvezeniePaletky : BOOL;
	END_STRUCT;
END_TYPE

(*//P3 - Leakage Test A//*)

TYPE
	P3_LeakageTestA_typ : 	STRUCT
		CMD : P3_LeakageTestA_CMD_typ;
		IN : P3_LeakageTestA_IN_typ;
		OUT : P3_LeakageTestA_OUT_typ;
		PAR : P3_LeakageTestA_PAR_typ;
		STAV : P3_LeakageTestA_STAV_typ;
		RFID_hlava : SickHeads;
		Automat : BOOL;
		Manual : BOOL;
		Reset : BOOL;
		KoniecCyklu : BOOL;
	END_STRUCT;
	P3_LeakageTestA_CMD_typ : 	STRUCT
		RR_HornyPritlak_VYSUN : BOOL;
		RR_HornyPritlak_ZASUN : BOOL;
		RR_VysunSpodneKopito : BOOL;
		RR_TestovaciaSekvencia_START : BOOL;
		RR_VysunCentrovanie : BOOL;
	END_STRUCT;
	P3_LeakageTestA_IN_typ : 	STRUCT
		NapajanieTestera_OK : BOOL;
		HornyPritlak_TlakOK : BOOL; (*S3.8*)
		HornyPritlak_PneuZamok_Odomknuty : BOOL; (*S3.9*)
		HornyPritlak_VYSUNUTY : BOOL; (*MS3_16*)
		HornyPritlak_ZASUNUTY : BOOL; (*MS3_15*)
		Centrovanie_VYSUNUTE : BOOL; (*IS3_36*)
		Centrovanie_ZASUNUTE : BOOL; (*IS3_37*)
		PritomnostKopita : BOOL; (*IS3_32*)
		Kopito_ZASUNUTE : BOOL; (*IS3_33*)
		VyrovnavaciTlak_OK : BOOL; (*S3_4 - IO-Link snímač*)
		Tester_TypKonektoru_4F : BOOL;
		Tester_TypKonektoru_5F_5H : BOOL;
	END_STRUCT;
	P3_LeakageTestA_OUT_typ : 	STRUCT
		HornyPritlak_VYSUN : BOOL; (*YV143_VT3*)
		HornyPritlak_ZASUN : BOOL; (*YV144_VT3*)
		PneuZamokZvonu_ODOMKNI : BOOL; (*YV145_VT3*)
		PneuZamokCentrovania_ODOMKNI : BOOL; (*YV168_VT3*)
		Kopito_VYSUN : BOOL; (*YV149_VT3*)
		Kopito_ZASUN : BOOL; (*YV150_VT3*)
		ZasunStoper : BOOL; (*YV115_VT3*)
		Centrovanie_VYSUN : BOOL; (*YV151_VT3*)
	END_STRUCT;
	P3_LeakageTestA_PAR_typ : 	STRUCT
		CisloPaletky_STRING : STRING[2];
		PrecitanyVyrovnavaciTlak : UINT; (*IO-Link snímač*)
		PreratanyVyrovnavaciTlak_Bar : REAL;
		CisloPaletky : USINT;
	END_STRUCT;
	P3_LeakageTestA_STAV_typ : 	STRUCT
		PoINIT : BOOL;
		PrebiehaVyvezeniePaletky : BOOL;
		Tester_ON : BOOL;
		RR_TestovaciaSekvencia_BUSY : BOOL;
	END_STRUCT;
END_TYPE

(*//P3 - Leakage Test B//*)

TYPE
	P3_LeakageTestB_typ : 	STRUCT
		CMD : P3_LeakageTestB_CMD_typ;
		IN : P3_LeakageTestB_IN_typ;
		OUT : P3_LeakageTestB_OUT_typ;
		PAR : P3_LeakageTestB_PAR_typ;
		STAV : P3_LeakageTestB_STAV_typ;
		RFID_hlava : SickHeads;
		Automat : BOOL;
		Manual : BOOL;
		Reset : BOOL;
		KoniecCyklu : BOOL;
	END_STRUCT;
	P3_LeakageTestB_CMD_typ : 	STRUCT
		RR_VysunSpodneKopito : BOOL;
		RR_TestovaciaSekvencia_START : BOOL;
		RR_VysunCentrovanie : BOOL;
		RR_HornyPritlak_VYSUN : BOOL;
		RR_HornyPritlak_ZASUN : BOOL;
	END_STRUCT;
	P3_LeakageTestB_IN_typ : 	STRUCT
		NapajanieTestera_OK : BOOL;
		HornyPritlak_TlakOK : BOOL; (*S3.10*)
		HornyPritlak_PneuZamok_Odomknuty : BOOL; (*S3.11*)
		HornyPritlak_VYSUNUTY : BOOL; (*MS3_18*)
		HornyPritlak_ZASUNUTY : BOOL; (*MS3_17*)
		Centrovanie_VYSUNUTE : BOOL; (*IS3_38*)
		Centrovanie_ZASUNUTE : BOOL; (*IS3_39*)
		PritomnostKopita : BOOL; (*IS3_34*)
		Kopito_ZASUNUTE : BOOL; (*IS3_35*)
		VyrovnavaciTlak_OK : BOOL; (*S3_5 - IO-Link snímač*)
		Tester_TypKonektoru_4F : BOOL;
		Tester_TypKonektoru_5F_5H : BOOL;
	END_STRUCT;
	P3_LeakageTestB_OUT_typ : 	STRUCT
		HornyPritlak_VYSUN : BOOL; (*YV146_VT3*)
		HornyPritlak_ZASUN : BOOL; (*YV147_VT3*)
		PneuZamokZvonu_ODOMKNI : BOOL; (*YV148_VT3*)
		PneuZamokCentrovania_ODOMKNI : BOOL; (*YV169_VT3*)
		Kopito_VYSUN : BOOL; (*YV153_VT3*)
		Kopito_ZASUN : BOOL; (*YV167_VT3*)
		ZasunStoper : BOOL; (*YV116_VT3*)
		Centrovanie_VYSUN : BOOL; (*YV154_VT3*)
	END_STRUCT;
	P3_LeakageTestB_PAR_typ : 	STRUCT
		CisloPaletky_STRING : STRING[2];
		PrecitanyVyrovnavaciTlak : UINT; (*IO-Link snímač*)
		PreratanyVyrovnavaciTlak_Bar : REAL;
		CisloPaletky : USINT;
	END_STRUCT;
	P3_LeakageTestB_STAV_typ : 	STRUCT
		PoINIT : BOOL;
		PrebiehaVyvezeniePaletky : BOOL;
		Tester_ON : BOOL;
		RR_TestovaciaSekvencia_BUSY : BOOL;
	END_STRUCT;
END_TYPE

(*//P3 - Zdvižka za Leakage Testom A//*)

TYPE
	P3_ZdvizkaZaLeakTestA_typ : 	STRUCT
		IN : P3_ZdvizkaZaLeakTestA_IN_typ;
		OUT : P3_ZdvizkaZaLeakTestA_OUT_typ;
		PAR : P3_ZdvizkaZaLeakTestA_PAR_typ;
		STAV : P3_ZdvizkaZaLeakTestA_STAV_typ;
		Automat : BOOL;
		Manual : BOOL;
		Reset : BOOL;
		KoniecCyklu : BOOL;
	END_STRUCT;
	P3_ZdvizkaZaLeakTestA_IN_typ : 	STRUCT
		PritomnostPaletky : BOOL; (*IS3_20*)
		PoziciaPaletky_OK : BOOL; (*IS3_19*)
		Zdvizka_HornaPoloha : BOOL; (*IS3_17*)
		Zdvizka_SpodnaPoloha : BOOL; (*IS3_16*)
		Zdvizka_StrednaPoloha : BOOL; (*IS3_18*)
		TlmicPaletky_ZASUNUTY : BOOL; (*MS3_2*)
	END_STRUCT;
	P3_ZdvizkaZaLeakTestA_OUT_typ : 	STRUCT
		Zdvizku_ZASUN : BOOL; (*YV117_VT3*)
		Zdvizku_VYSUN : BOOL; (*YV118_VT3*)
		TlmicPaletky_VYSUN : BOOL; (*YV119_VT3*)
		TlmicPaletky_ZASUN : BOOL; (*YV120_VT3*)
	END_STRUCT;
	P3_ZdvizkaZaLeakTestA_PAR_typ : 	STRUCT
		New_Member : USINT;
	END_STRUCT;
	P3_ZdvizkaZaLeakTestA_STAV_typ : 	STRUCT
		PoINIT : BOOL;
		PrebiehaVyvezeniePaletkyNaTratA : BOOL;
		PrebiehaVyvezeniePaletkyNaTratB : BOOL;
	END_STRUCT;
END_TYPE

(*//P3 - Zdvižka za Leakage Testom B//*)

TYPE
	P3_ZdvizkaZaLeakTestB_typ : 	STRUCT
		IN : P3_ZdvizkaZaLeakTestB_IN_typ;
		OUT : P3_ZdvizkaZaLeakTestB_OUT_typ;
		PAR : P3_ZdvizkaZaLeakTestB_PAR_typ;
		STAV : P3_ZdvizkaZaLeakTestB_STAV_typ;
		Automat : BOOL;
		Manual : BOOL;
		Reset : BOOL;
		KoniecCyklu : BOOL;
	END_STRUCT;
	P3_ZdvizkaZaLeakTestB_IN_typ : 	STRUCT
		PritomnostPaletky : BOOL; (*IS3_25*)
		PoziciaPaletky_OK : BOOL; (*IS3_24*)
		Zdvizka_HornaPoloha : BOOL; (*IS3_22*)
		Zdvizka_SpodnaPoloha : BOOL; (*IS3_21*)
		Zdvizka_StrednaPoloha : BOOL; (*IS3_23*)
		TlmicPaletky_ZASUNUTY : BOOL; (*MS3_3*)
	END_STRUCT;
	P3_ZdvizkaZaLeakTestB_OUT_typ : 	STRUCT
		Zdvizku_ZASUN : BOOL; (*YV121_VT3*)
		Zdvizku_VYSUN : BOOL; (*YV122_VT3*)
		TlmicPaletky_VYSUN : BOOL; (*YV123_VT3*)
		TlmicPaletky_ZASUN : BOOL; (*YV124_VT3*)
	END_STRUCT;
	P3_ZdvizkaZaLeakTestB_PAR_typ : 	STRUCT
		New_Member : USINT;
	END_STRUCT;
	P3_ZdvizkaZaLeakTestB_STAV_typ : 	STRUCT
		PoINIT : BOOL;
		PrebiehaVyvezeniePaletkyNaTratA : BOOL;
		PrebiehaVyvezeniePaletkyNaTratB : BOOL;
	END_STRUCT;
END_TYPE

(***********************************Pracovisko 4****************************************************************)

TYPE
	P4_Pracovisko_typ : 	STRUCT
		IN : P4_PracoviskoIN_typ;
		OUT : P4_PracoviskoOUT_typ;
		PAR : P4_PracoviskoPAR_typ;
		STAV : P4_PracoviskoSTAV_typ;
		COM_Weidmuller : P4_COM_Weidmuller_typ;
		COM_Festo : P4_COM_Festo_typ;
		COM_VentilovyTerminal : ARRAY[0..9]OF USINT;
		Automat : BOOL;
		Manual : BOOL;
		Reset : BOOL;
		KoniecCyklu : BOOL;
		KoniecVyroby : BOOL;
	END_STRUCT;
	P4_PracoviskoIN_typ : 	STRUCT
		TlakVzduchu_OK : BOOL; (*S4_5*)
		ModulWeidmuller_IO_KomOK : BOOL;
		VentilovyTerminal_KomOK : BOOL;
		ModulFesto_IO_KomOK : BOOL;
		ServoZdvihuVytahu_KomOK : BOOL;
		ServoZdvihuAplikEtikiet_KomOK : BOOL;
		SmartKamera14_KomOK : BOOL;
		PredneDvere_PritomnostAdaptera : BOOL; (*EZ 4.1*)
		ZadneDvere_PritomnostAdaptera : BOOL; (*EZ 4.2*)
	END_STRUCT;
	P4_PracoviskoOUT_typ : 	STRUCT
		Majak_ZeleneSvetlo_ON : BOOL;
		Majak_OranzoveSvetlo_ON : BOOL;
		Majak_CerveneSvetlo_ON : BOOL;
		Majak_Hukacka_ON : BOOL;
		OsvetlenieBunky_ON : BOOL;
		Osvetlenie_CAM16_ON : BOOL;
		Osvetlenie_CAM15_ON : BOOL;
		ZdvizkyPneuZamok_ODOMKNI : BOOL; (*YV174_VT4*)
		PredneDvere_ZAMKNI : BOOL; (*EZ 4.1*)
		ZadneDvere_ZAMKNI : BOOL; (*EZ 4.2*)
	END_STRUCT;
	P4_PracoviskoPAR_typ : 	STRUCT
		New_Member : USINT;
	END_STRUCT;
	P4_PracoviskoSTAV_typ : 	STRUCT
		Automat : BOOL;
		Manual : BOOL;
		PoINIT : BOOL;
		READY : BOOL;
		PORUCHA : BOOL;
		HardwareBunky_OK : BOOL;
		HardwareVytahu_OK : BOOL;
		UkoncenieCyklu_BUSY : BOOL;
		Porucha_ST1 : BOOL; (*Final test A*)
		Porucha_ST2 : BOOL; (*Final test B*)
		Porucha_ST3 : BOOL; (*Zdvizka za Final testom A*)
		Porucha_ST4 : BOOL; (*Zdvizka za Final testom B*)
		Porucha_ST5 : BOOL; (*Etiketovanie*)
		Porucha_ST6 : BOOL; (*Výstupný výťah*)
		FunkcnyTestA_Zasunuty : BOOL;
		FunkcnyTestB_Zasunuty : BOOL;
	END_STRUCT;
	P4_COM_Weidmuller_typ : 	STRUCT
		AB4_2_8DI : USINT;
		AB4_3_8DI : USINT;
		AB4_4_8DI : USINT;
		AB4_5_8DO : USINT;
		AB4_6_8DO : USINT;
		AB4_8_8DO : USINT;
	END_STRUCT;
	P4_COM_Festo_typ : 	STRUCT
		DM4_1_4DI : ARRAY[0..3]OF BOOL;
		DM4_1_4DO : ARRAY[0..3]OF BOOL;
		DI4_1_8DI : ARRAY[0..7]OF BOOL;
		DI4_2_8DI : ARRAY[0..7]OF BOOL;
		DI4_3_8DI : ARRAY[0..7]OF BOOL;
		DI4_4_8DI : ARRAY[0..7]OF BOOL;
		DI4_5_8DI : ARRAY[0..7]OF BOOL;
		DS4_1_Port0_IN : ARRAY[0..31]OF USINT;
		DS4_1_Port0_OUT : ARRAY[0..31]OF USINT;
		DS4_1_Port1_IN : ARRAY[0..31]OF USINT;
		DS4_1_Port1_OUT : ARRAY[0..31]OF USINT;
		DS4_1_Port2_IN : ARRAY[0..31]OF USINT;
		DS4_1_Port2_OUT : ARRAY[0..31]OF USINT;
		DS4_2_Port0_IN : ARRAY[0..15]OF USINT;
		DS4_2_Port0_OUT : ARRAY[0..15]OF USINT;
		DS4_2_Port1_IN : ARRAY[0..31]OF USINT;
		DS4_2_Port1_OUT : ARRAY[0..31]OF USINT;
	END_STRUCT;
END_TYPE

(*//P4 - Dopravníky//*)

TYPE
	P4_Dopravniky_typ : 	STRUCT
		IN : P4_Dopravniky_IN_typ;
		OUT : P4_Dopravniky_OUT_typ;
		PAR : P4_Dopravniky_PAR_typ;
		STAV : P4_Dopravniky_STAV_typ;
		Automat : BOOL;
		Manual : BOOL;
		Reset : BOOL;
		KoniecCyklu : BOOL;
	END_STRUCT;
	P4_Dopravniky_IN_typ : 	STRUCT
		StavRiadPredDopravBunky_READY : BOOL; (*M4_4*)
		StavRiadZadnDopravBunky_READY : BOOL; (*M4_6*)
		StavRiadeniaPriecnDoprav_READY : BOOL; (*M4_5*)
		StavRiadeniaVratnehoDoprav_READY : BOOL; (*M4_7*)
		TeplotaMotoraPredDopravBunky_OK : BOOL; (*M4_4*)
		TeplotaMotoraZadnDopravBunky_OK : BOOL; (*M4_6*)
		TeplotaMotoraPriecnDoprav_OK : BOOL; (*M4_5*)
		TeplotaMotoraVratnehoDoprav_OK : BOOL; (*M4_7*)
	END_STRUCT;
	P4_Dopravniky_OUT_typ : 	STRUCT
		VratnyDopravnik_ON : BOOL; (*M4_7*)
		PrednyDopravnikBunky_ON : BOOL; (*M4_4*)
		ZadnyDopravnikBunky_ON : BOOL; (*M4_6*)
		PriecnyDopravnik_VPRED : BOOL; (*M4_5 - Smerom na trať A*)
	END_STRUCT;
	P4_Dopravniky_PAR_typ : 	STRUCT
		New_Member : USINT;
	END_STRUCT;
	P4_Dopravniky_STAV_typ : 	STRUCT
		PoINIT : BOOL;
	END_STRUCT;
END_TYPE
```
